LIN {X 0,Y 455.491,Z 844.733,A -85,B 0,C 180,E1 19302.236,E2 19302.236} C_VEL
LIN {X 0,Y 459.84,Z 821.771,A -85,B 0,C 180,E1 19301.253,E2 19301.253} C_VEL
LIN {X 0,Y 463.636,Z 798.381,A -85,B 0,C 180,E1 19300.452,E2 19300.452} C_VEL
LIN {X 0,Y 466.606,Z 774.028,A -85,B 0,C 180,E1 19299.835,E2 19299.835} C_VEL
LIN {X 0,Y 468.518,Z 750.577,A -85,B 0,C 180,E1 19299.385,E2 19299.385} C_VEL
LIN {X 0,Y 481.73,Z 500.688,A -85,B 0,C 180,E1 19295.435,E2 19295.435} C_VEL
LIN {X 0,Y 482.067,Z 491.701,A -85,B 0,C 180,E1 19295.268,E2 19295.268} C_VEL
LIN {X 0,Y 472.219,Z 474.079,A -85,B 0,C 180,E1 19293.15,E2 19293.15} C_VEL
LIN {X 0,Y 462.43,Z 457.753,A -85,B 0,C 180,E1 19290.861,E2 19290.861} C_VEL
LIN {X 0,Y 452.462,Z 442.354,A -85,B 0,C 180,E1 19288.296,E2 19288.296} C_VEL
LIN {X 0,Y 445.961,Z 432.998,A -85,B 0,C 180,E1 19286.463,E2 19286.463} C_VEL
LIN {X 0,Y 439.102,Z 423.302,A -85,B 0,C 180,E1 19284.341,E2 19284.341} C_VEL
LIN {X 0,Y 433.648,Z 416.334,A -85,B 0,C 180,E1 19282.505,E2 19282.505} C_VEL
LIN {X 0,Y 429.886,Z 411.664,A -85,B 0,C 180,E1 19281.132,E2 19281.132} C_VEL
LIN {X 0,Y 425.512,Z 406.796,A -85,B 0,C 180,E1 19279.421,E2 19279.421} C_VEL
LIN {X 0,Y 424.17,Z 404.903,A -85,B 0,C 180,E1 19278.841,E2 19278.841} C_VEL
LIN {X 0,Y 420.773,Z 401.5,A -85,B 0,C 180,E1 19277.351,E2 19277.351} C_VEL
LIN {X 0,Y 419.067,Z 398.833,A -85,B 0,C 180,E1 19276.495,E2 19276.495} C_VEL
LIN {X 0,Y 415.64,Z 396.018,A -85,B 0,C 180,E1 19274.774,E2 19274.774} C_VEL
LIN {X 0,Y 413.682,Z 392.463,A -85,B 0,C 180,E1 19273.56,E2 19273.56} C_VEL
LIN {X 0,Y 409.982,Z 390.014,A -85,B 0,C 180,E1 19271.251,E2 19271.251} C_VEL
LIN {X 0,Y 408.148,Z 386.758,A -85,B 0,C 180,E1 19269.732,E2 19269.732} C_VEL
LIN {X 0,Y 407.71,Z 385.774,A -85,B 0,C 180,E1 19269.315,E2 19269.315} C_VEL
LIN {X 0,Y 403.812,Z 383.595,A -85,B 0,C 180,E1 19265.399,E2 19265.399} C_VEL
LIN {X 0,Y 401.716,Z 379.418,A -85,B 0,C 180,E1 19259.857,E2 19259.857} C_VEL
LIN {X 0,Y 401.699,Z 379.301,A -85,B 0,C 180,E1 19258.003,E2 19258.003} C_VEL
LIN {X 0,Y 402.926,Z 382.497,A -85,B 0,C 180,E1 19253.588,E2 19253.588} C_VEL
LIN {X 0,Y 406.71,Z 385.47,A -85,B 0,C 180,E1 19249.088,E2 19249.088} C_VEL
LIN {X 0,Y 407.878,Z 386.044,A -85,B 0,C 180,E1 19248.116,E2 19248.116} C_VEL
LIN {X 0,Y 409.365,Z 389.184,A -85,B 0,C 180,E1 19246.798,E2 19246.798} C_VEL
LIN {X 0,Y 412.3,Z 391.844,A -85,B 0,C 180,E1 19244.816,E2 19244.816} C_VEL
LIN {X 0,Y 413.753,Z 392.667,A -85,B 0,C 180,E1 19243.972,E2 19243.972} C_VEL
LIN {X 0,Y 416.055,Z 396.475,A -85,B 0,C 180,E1 19242.583,E2 19242.583} C_VEL
LIN {X 0,Y 419.443,Z 399.307,A -85,B 0,C 180,E1 19240.902,E2 19240.902} C_VEL
LIN {X 0,Y 422.238,Z 403.299,A -85,B 0,C 180,E1 19239.556,E2 19239.556} C_VEL
LIN {X 0,Y 424.839,Z 405.657,A -85,B 0,C 180,E1 19238.459,E2 19238.459} C_VEL
LIN {X 0,Y 428.113,Z 409.894,A -85,B 0,C 180,E1 19237.115,E2 19237.115} C_VEL
LIN {X 0,Y 430.045,Z 411.854,A -85,B 0,C 180,E1 19236.391,E2 19236.391} C_VEL
LIN {X 0,Y 433.924,Z 416.564,A -85,B 0,C 180,E1 19234.986,E2 19234.986} C_VEL
LIN {X 0,Y 439.996,Z 424.177,A -85,B 0,C 180,E1 19232.967,E2 19232.967} C_VEL
LIN {X 0,Y 444.51,Z 429.966,A -85,B 0,C 180,E1 19231.585,E2 19231.585} C_VEL
LIN {X 0,Y 451.641,Z 439.191,A -85,B 0,C 180,E1 19229.573,E2 19229.573} C_VEL
LIN {X 0,Y 461.95,Z 453.355,A -85,B 0,C 180,E1 19226.944,E2 19226.944} C_VEL
LIN {X 0,Y 473.346,Z 470.153,A -85,B 0,C 180,E1 19224.337,E2 19224.337} C_VEL
LIN {X 0,Y 482.433,Z 484.639,A -85,B 0,C 180,E1 19222.43,E2 19222.43} C_VEL
LIN {X 0,Y 468.967,Z 736.517,A -85,B 0,C 180,E1 19218.449,E2 19218.449} C_VEL
LIN {X 0,Y 467.166,Z 758.61,A -85,B 0,C 180,E1 19218.013,E2 19218.013} C_VEL
LIN {X 0,Y 464.253,Z 783.344,A -85,B 0,C 180,E1 19217.35,E2 19217.35} C_VEL
LIN {X 0,Y 460.975,Z 804.43,A -85,B 0,C 180,E1 19216.605,E2 19216.605} C_VEL
LIN {X 0,Y 457.064,Z 825.889,A -85,B 0,C 180,E1 19215.672,E2 19215.672} C_VEL
LIN {X 0,Y 452.059,Z 849.09,A -85,B 0,C 180,E1 19214.422,E2 19214.422} C_VEL
LIN {X 0,Y 447.255,Z 868.657,A -85,B 0,C 180,E1 19213.165,E2 19213.165} C_VEL
LIN {X 0,Y 441.166,Z 891.084,A -85,B 0,C 180,E1 19211.438,E2 19211.438} C_VEL
LIN {X 0,Y 435.995,Z 908.438,A -85,B 0,C 180,E1 19209.866,E2 19209.866} C_VEL
LIN {X 0,Y 429.83,Z 928.005,A -85,B 0,C 180,E1 19207.804,E2 19207.804} C_VEL
LIN {X 0,Y 424.092,Z 945.022,A -85,B 0,C 180,E1 19205.687,E2 19205.687} C_VEL
LIN {X 0,Y 418.144,Z 962.284,A -85,B 0,C 180,E1 19203.202,E2 19203.202} C_VEL
LIN {X 0,Y 412.713,Z 977.598,A -85,B 0,C 180,E1 19200.582,E2 19200.582} C_VEL
LIN {X 0,Y 407.773,Z 991.832,A -85,B 0,C 180,E1 19197.768,E2 19197.768} C_VEL
LIN {X 0,Y 403.388,Z 1004.565,A -85,B 0,C 180,E1 19194.765,E2 19194.765} C_VEL
LIN {X 0,Y 399.844,Z 1015.636,A -85,B 0,C 180,E1 19191.722,E2 19191.722} C_VEL
LIN {X 0,Y 396.862,Z 1025.775,A -85,B 0,C 180,E1 19188.357,E2 19188.357} C_VEL
LIN {X 0,Y 394.876,Z 1033.558,A -85,B 0,C 180,E1 19185.256,E2 19185.256} C_VEL
LIN {X 0,Y 393.323,Z 1040.946,A -85,B 0,C 180,E1 19181.586,E2 19181.586} C_VEL
LIN {X 0,Y 392.551,Z 1045.732,A -85,B 0,C 180,E1 19178.496,E2 19178.496} C_VEL
LIN {X 0,Y 392.145,Z 1049.646,A -85,B 0,C 180,E1 19175.12,E2 19175.12} C_VEL
LIN {X 0,Y 391.997,Z 1051.962,A -85,B 0,C 180,E1 19171.754,E2 19171.754} C_VEL
LIN {X 0,Y 391.965,Z 1052.864,A -85,B 0,C 180,E1 19168.977,E2 19168.977} C_VEL
LIN {X 0,Y 391.973,Z 1052.777,A -85,B 0,C 180,E1 19165.904,E2 19165.904} C_VEL
LIN {X 0,Y 392.058,Z 1051.214,A -85,B 0,C 180,E1 19162.379,E2 19162.379} C_VEL
LIN {X 0,Y 392.307,Z 1048.524,A -85,B 0,C 180,E1 19159.277,E2 19159.277} C_VEL
LIN {X 0,Y 392.861,Z 1044.661,A -85,B 0,C 180,E1 19156.158,E2 19156.158} C_VEL
LIN {X 0,Y 393.592,Z 1040.768,A -85,B 0,C 180,E1 19153.731,E2 19153.731} C_VEL
LIN {X 0,Y 393.032,Z 1038.922,A -85,B 0,C 180,E1 19152.636,E2 19152.636} C_VEL
LIN {X 0,Y 388.297,Z 1033.538,A -85,B 0,C 180,E1 19149.698,E2 19149.698} C_VEL
LIN {X 0,Y 388.161,Z 1031.488,A -85,B 0,C 180,E1 19148.76,E2 19148.76} C_VEL
LIN {X 0,Y 391.208,Z 1021.724,A -85,B 0,C 180,E1 19145.057,E2 19145.057} C_VEL
LIN {X 0,Y 394.53,Z 1012.11,A -85,B 0,C 180,E1 19142.04,E2 19142.04} C_VEL
LIN {X 0,Y 399.372,Z 999.124,A -85,B 0,C 180,E1 19138.617,E2 19138.617} C_VEL
LIN {X 0,Y 404.183,Z 986.584,A -85,B 0,C 180,E1 19135.836,E2 19135.836} C_VEL
LIN {X 0,Y 410.106,Z 971.471,A -85,B 0,C 180,E1 19132.971,E2 19132.971} C_VEL
LIN {X 0,Y 416.021,Z 956.003,A -85,B 0,C 180,E1 19130.49,E2 19130.49} C_VEL
LIN {X 0,Y 422.663,Z 938.384,A -85,B 0,C 180,E1 19128.063,E2 19128.063} C_VEL
LIN {X 0,Y 428.961,Z 920.629,A -85,B 0,C 180,E1 19126.003,E2 19126.003} C_VEL
LIN {X 0,Y 435.548,Z 901.209,A -85,B 0,C 180,E1 19124.065,E2 19124.065} C_VEL
LIN {X 0,Y 441.835,Z 880.625,A -85,B 0,C 180,E1 19122.35,E2 19122.35} C_VEL
LIN {X 0,Y 447.423,Z 860.804,A -85,B 0,C 180,E1 19120.944,E2 19120.944} C_VEL
LIN {X 0,Y 453.017,Z 838.232,A -85,B 0,C 180,E1 19119.619,E2 19119.619} C_VEL
LIN {X 0,Y 457.191,Z 818.895,A -85,B 0,C 180,E1 19118.669,E2 19118.669} C_VEL
LIN {X 0,Y 461.767,Z 793.938,A -85,B 0,C 180,E1 19117.68,E2 19117.68} C_VEL
LIN {X 0,Y 464.905,Z 772.264,A -85,B 0,C 180,E1 19117.014,E2 19117.014} C_VEL
LIN {X 0,Y 467.655,Z 747.34,A -85,B 0,C 180,E1 19116.439,E2 19116.439} C_VEL
LIN {X 0,Y 471.279,Z 687.121,A -85,B 0,C 180,E1 19115.457,E2 19115.457} C_VEL
LIN {X 0,Y 482.561,Z 491.611,A -85,B 0,C 180,E1 19112.355,E2 19112.355} C_VEL
LIN {X 0,Y 471.614,Z 474.658,A -85,B 0,C 180,E1 19109.778,E2 19109.778} C_VEL
LIN {X 0,Y 462.04,Z 460.876,A -85,B 0,C 180,E1 19107.274,E2 19107.274} C_VEL
LIN {X 0,Y 454.319,Z 450.447,A -85,B 0,C 180,E1 19105.032,E2 19105.032} C_VEL
LIN {X 0,Y 447.642,Z 441.602,A -85,B 0,C 180,E1 19102.871,E2 19102.871} C_VEL
LIN {X 0,Y 443.202,Z 436.029,A -85,B 0,C 180,E1 19101.299,E2 19101.299} C_VEL
LIN {X 0,Y 439.218,Z 430.987,A -85,B 0,C 180,E1 19099.759,E2 19099.759} C_VEL
LIN {X 0,Y 435.448,Z 426.19,A -85,B 0,C 180,E1 19098.163,E2 19098.163} C_VEL
LIN {X 0,Y 431.395,Z 421.665,A -85,B 0,C 180,E1 19096.287,E2 19096.287} C_VEL
LIN {X 0,Y 430.163,Z 419.832,A -85,B 0,C 180,E1 19095.643,E2 19095.643} C_VEL
LIN {X 0,Y 426.685,Z 416.352,A -85,B 0,C 180,E1 19093.76,E2 19093.76} C_VEL
LIN {X 0,Y 425.161,Z 413.779,A -85,B 0,C 180,E1 19092.772,E2 19092.772} C_VEL
LIN {X 0,Y 421.812,Z 411.007,A -85,B 0,C 180,E1 19090.517,E2 19090.517} C_VEL
LIN {X 0,Y 419.877,Z 407.432,A -85,B 0,C 180,E1 19088.767,E2 19088.767} C_VEL
LIN {X 0,Y 415.834,Z 404.429,A -85,B 0,C 180,E1 19083.999,E2 19083.999} C_VEL
LIN {X 0,Y 414.742,Z 401.753,A -85,B 0,C 180,E1 19080.138,E2 19080.138} C_VEL
LIN {X 0,Y 414.717,Z 401.619,A -85,B 0,C 180,E1 19078.618,E2 19078.618} C_VEL
LIN {X 0,Y 415.242,Z 403.337,A -85,B 0,C 180,E1 19075.719,E2 19075.719} C_VEL
LIN {X 0,Y 419.25,Z 407.195,A -85,B 0,C 180,E1 19070.112,E2 19070.112} C_VEL
LIN {X 0,Y 420.088,Z 407.737,A -85,B 0,C 180,E1 19069.37,E2 19069.37} C_VEL
LIN {X 0,Y 422.241,Z 411.567,A -85,B 0,C 180,E1 19067.486,E2 19067.486} C_VEL
LIN {X 0,Y 425.517,Z 414.256,A -85,B 0,C 180,E1 19065.333,E2 19065.333} C_VEL
LIN {X 0,Y 428.154,Z 418.196,A -85,B 0,C 180,E1 19063.725,E2 19063.725} C_VEL
LIN {X 0,Y 430.667,Z 420.442,A -85,B 0,C 180,E1 19062.433,E2 19062.433} C_VEL
LIN {X 0,Y 434.083,Z 424.878,A -85,B 0,C 180,E1 19060.768,E2 19060.768} C_VEL
LIN {X 0,Y 435.806,Z 426.713,A -85,B 0,C 180,E1 19060.01,E2 19060.01} C_VEL
LIN {X 0,Y 439.552,Z 431.305,A -85,B 0,C 180,E1 19058.446,E2 19058.446} C_VEL
LIN {X 0,Y 446.538,Z 441.039,A -85,B 0,C 180,E1 19055.809,E2 19055.809} C_VEL
LIN {X 0,Y 454.673,Z 452.672,A -85,B 0,C 180,E1 19053.133,E2 19053.133} C_VEL
LIN {X 0,Y 464.779,Z 468.395,A -85,B 0,C 180,E1 19050.201,E2 19050.201} C_VEL
LIN {X 0,Y 473.883,Z 483.545,A -85,B 0,C 180,E1 19047.842,E2 19047.842} C_VEL
LIN {X 0,Y 482.418,Z 498.724,A -85,B 0,C 180,E1 19045.816,E2 19045.816} C_VEL
LIN {X 0,Y 468.053,Z 748.938,A -85,B 0,C 180,E1 19041.855,E2 19041.855} C_VEL
LIN {X 0,Y 465.972,Z 773.134,A -85,B 0,C 180,E1 19041.396,E2 19041.396} C_VEL
LIN {X 0,Y 462.858,Z 797.389,A -85,B 0,C 180,E1 19040.795,E2 19040.795} C_VEL
LIN {X 0,Y 458.752,Z 821.123,A -85,B 0,C 180,E1 19039.997,E2 19039.997} C_VEL
LIN {X 0,Y 454.683,Z 841.259,A -85,B 0,C 180,E1 19039.156,E2 19039.156} C_VEL
LIN {X 0,Y 449.116,Z 864.849,A -85,B 0,C 180,E1 19037.934,E2 19037.934} C_VEL
LIN {X 0,Y 444.065,Z 883.795,A -85,B 0,C 180,E1 19036.754,E2 19036.754} C_VEL
LIN {X 0,Y 437.897,Z 904.941,A -85,B 0,C 180,E1 19035.198,E2 19035.198} C_VEL
LIN {X 0,Y 431.615,Z 924.469,A -85,B 0,C 180,E1 19033.475,E2 19033.475} C_VEL
LIN {X 0,Y 425.219,Z 943.337,A -85,B 0,C 180,E1 19031.538,E2 19031.538} C_VEL
LIN {X 0,Y 418.497,Z 961.862,A -85,B 0,C 180,E1 19029.275,E2 19029.275} C_VEL
LIN {X 0,Y 412.462,Z 978.197,A -85,B 0,C 180,E1 19026.956,E2 19026.956} C_VEL
LIN {X 0,Y 406.308,Z 994.527,A -85,B 0,C 180,E1 19024.221,E2 19024.221} C_VEL
LIN {X 0,Y 401.467,Z 1007.481,A -85,B 0,C 180,E1 19021.703,E2 19021.703} C_VEL
LIN {X 0,Y 396.129,Z 1022.244,A -85,B 0,C 180,E1 19018.329,E2 19018.329} C_VEL
LIN {X 0,Y 392.382,Z 1033.25,A -85,B 0,C 180,E1 19015.348,E2 19015.348} C_VEL
LIN {X 0,Y 388.944,Z 1044.487,A -85,B 0,C 180,E1 19011.727,E2 19011.727} C_VEL
LIN {X 0,Y 386.8,Z 1052.635,A -85,B 0,C 180,E1 19008.54,E2 19008.54} C_VEL
LIN {X 0,Y 385.198,Z 1060.295,A -85,B 0,C 180,E1 19004.891,E2 19004.891} C_VEL
LIN {X 0,Y 384.382,Z 1065.649,A -85,B 0,C 180,E1 19001.554,E2 19001.554} C_VEL
LIN {X 0,Y 384.037,Z 1069.516,A -85,B 0,C 180,E1 18998.384,E2 18998.384} C_VEL
LIN {X 0,Y 383.949,Z 1072.401,A -85,B 0,C 180,E1 18994.78,E2 18994.78} C_VEL
LIN {X 0,Y 383.953,Z 1073.541,A -85,B 0,C 180,E1 18991.642,E2 18991.642} C_VEL
LIN {X 0,Y 383.963,Z 1073.547,A -85,B 0,C 180,E1 18988.806,E2 18988.806} C_VEL
LIN {X 0,Y 383.948,Z 1072.419,A -85,B 0,C 180,E1 18985.669,E2 18985.669} C_VEL
LIN {X 0,Y 384.004,Z 1069.534,A -85,B 0,C 180,E1 18982.068,E2 18982.068} C_VEL
LIN {X 0,Y 384.28,Z 1065.866,A -85,B 0,C 180,E1 18979.05,E2 18979.05} C_VEL
LIN {X 0,Y 384.979,Z 1060.531,A -85,B 0,C 180,E1 18975.715,E2 18975.715} C_VEL
LIN {X 0,Y 386.406,Z 1052.891,A -85,B 0,C 180,E1 18972.065,E2 18972.065} C_VEL
LIN {X 0,Y 388.362,Z 1044.717,A -85,B 0,C 180,E1 18968.872,E2 18968.872} C_VEL
LIN {X 0,Y 391.549,Z 1033.43,A -85,B 0,C 180,E1 18965.241,E2 18965.241} C_VEL
LIN {X 0,Y 394.875,Z 1022.921,A -85,B 0,C 180,E1 18962.394,E2 18962.394} C_VEL
LIN {X 0,Y 399.705,Z 1008.63,A -85,B 0,C 180,E1 18959.098,E2 18959.098} C_VEL
LIN {X 0,Y 404.296,Z 995.515,A -85,B 0,C 180,E1 18956.529,E2 18956.529} C_VEL
LIN {X 0,Y 409.981,Z 979.623,A -85,B 0,C 180,E1 18953.828,E2 18953.828} C_VEL
LIN {X 0,Y 415.936,Z 962.527,A -85,B 0,C 180,E1 18951.379,E2 18951.379} C_VEL
LIN {X 0,Y 422.291,Z 944.111,A -85,B 0,C 180,E1 18949.104,E2 18949.104} C_VEL
LIN {X 0,Y 428.466,Z 924.968,A -85,B 0,C 180,E1 18947.119,E2 18947.119} C_VEL
LIN {X 0,Y 434.363,Z 905.758,A -85,B 0,C 180,E1 18945.404,E2 18945.404} C_VEL
LIN {X 0,Y 440.427,Z 884.078,A -85,B 0,C 180,E1 18943.785,E2 18943.785} C_VEL
LIN {X 0,Y 445.338,Z 864.832,A -85,B 0,C 180,E1 18942.571,E2 18942.571} C_VEL
LIN {X 0,Y 450.75,Z 840.786,A -85,B 0,C 180,E1 18941.316,E2 18941.316} C_VEL
LIN {X 0,Y 454.679,Z 820.431,A -85,B 0,C 180,E1 18940.457,E2 18940.457} C_VEL
LIN {X 0,Y 458.627,Z 796.402,A -85,B 0,C 180,E1 18939.647,E2 18939.647} C_VEL
LIN {X 0,Y 461.517,Z 772.739,A -85,B 0,C 180,E1 18939.057,E2 18939.057} C_VEL
LIN {X 0,Y 463.533,Z 747.792,A -85,B 0,C 180,E1 18938.583,E2 18938.583} C_VEL
LIN {X 0,Y 477.177,Z 497.517,A -85,B 0,C 180,E1 18934.61,E2 18934.61} C_VEL
LIN {X 0,Y 477.146,Z 495.381,A -85,B 0,C 180,E1 18934.551,E2 18934.551} C_VEL
LIN {X 0,Y 468.133,Z 479.157,A -85,B 0,C 180,E1 18932.547,E2 18932.547} C_VEL
LIN {X 0,Y 458.488,Z 462.849,A -85,B 0,C 180,E1 18930.214,E2 18930.214} C_VEL
LIN {X 0,Y 448.517,Z 447.367,A -85,B 0,C 180,E1 18927.554,E2 18927.554} C_VEL
LIN {X 0,Y 440.843,Z 436.152,A -85,B 0,C 180,E1 18925.276,E2 18925.276} C_VEL
LIN {X 0,Y 435.436,Z 428.576,A -85,B 0,C 180,E1 18923.515,E2 18923.515} C_VEL
LIN {X 0,Y 431.436,Z 423.529,A -85,B 0,C 180,E1 18922.124,E2 18922.124} C_VEL
LIN {X 0,Y 427.082,Z 418.165,A -85,B 0,C 180,E1 18920.488,E2 18920.488} C_VEL
LIN {X 0,Y 423.465,Z 413.928,A -85,B 0,C 180,E1 18919.017,E2 18919.017} C_VEL
LIN {X 0,Y 422.283,Z 412.371,A -85,B 0,C 180,E1 18918.499,E2 18918.499} C_VEL
LIN {X 0,Y 418.833,Z 408.657,A -85,B 0,C 180,E1 18916.933,E2 18916.933} C_VEL
LIN {X 0,Y 417.554,Z 406.557,A -85,B 0,C 180,E1 18916.271,E2 18916.271} C_VEL
LIN {X 0,Y 414.063,Z 403.556,A -85,B 0,C 180,E1 18914.474,E2 18914.474} C_VEL
LIN {X 0,Y 412.008,Z 400.163,A -85,B 0,C 180,E1 18913.187,E2 18913.187} C_VEL
LIN {X 0,Y 408.446,Z 397.48,A -85,B 0,C 180,E1 18910.865,E2 18910.865} C_VEL
LIN {X 0,Y 406.632,Z 393.911,A -85,B 0,C 180,E1 18909.269,E2 18909.269} C_VEL
LIN {X 0,Y 402.105,Z 390.661,A -85,B 0,C 180,E1 18904.278,E2 18904.278} C_VEL
LIN {X 0,Y 400.727,Z 387.333,A -85,B 0,C 180,E1 18899.714,E2 18899.714} C_VEL
LIN {X 0,Y 400.721,Z 387.274,A -85,B 0,C 180,E1 18897.998,E2 18897.998} C_VEL
LIN {X 0,Y 401.95,Z 390.495,A -85,B 0,C 180,E1 18893.573,E2 18893.573} C_VEL
LIN {X 0,Y 405.751,Z 393.425,A -85,B 0,C 180,E1 18889.062,E2 18889.062} C_VEL
LIN {X 0,Y 406.606,Z 393.952,A -85,B 0,C 180,E1 18888.331,E2 18888.331} C_VEL
LIN {X 0,Y 408.39,Z 397.344,A -85,B 0,C 180,E1 18886.766,E2 18886.766} C_VEL
LIN {X 0,Y 411.352,Z 399.841,A -85,B 0,C 180,E1 18884.78,E2 18884.78} C_VEL
LIN {X 0,Y 412.319,Z 400.519,A -85,B 0,C 180,E1 18884.204,E2 18884.204} C_VEL
LIN {X 0,Y 414.954,Z 404.57,A -85,B 0,C 180,E1 18882.615,E2 18882.615} C_VEL
LIN {X 0,Y 417.856,Z 407.066,A -85,B 0,C 180,E1 18881.153,E2 18881.153} C_VEL
LIN {X 0,Y 420.843,Z 411.141,A -85,B 0,C 180,E1 18879.703,E2 18879.703} C_VEL
LIN {X 0,Y 423.031,Z 413.181,A -85,B 0,C 180,E1 18878.763,E2 18878.763} C_VEL
LIN {X 0,Y 426.507,Z 417.6,A -85,B 0,C 180,E1 18877.316,E2 18877.316} C_VEL
LIN {X 0,Y 428.237,Z 419.511,A -85,B 0,C 180,E1 18876.65,E2 18876.65} C_VEL
LIN {X 0,Y 433.3,Z 425.813,A -85,B 0,C 180,E1 18874.801,E2 18874.801} C_VEL
LIN {X 0,Y 438.073,Z 431.845,A -85,B 0,C 180,E1 18873.206,E2 18873.206} C_VEL
LIN {X 0,Y 444.947,Z 440.653,A -85,B 0,C 180,E1 18871.108,E2 18871.108} C_VEL
LIN {X 0,Y 455.338,Z 454.837,A -85,B 0,C 180,E1 18868.269,E2 18868.269} C_VEL
LIN {X 0,Y 465.733,Z 470.04,A -85,B 0,C 180,E1 18865.734,E2 18865.734} C_VEL
LIN {X 0,Y 476.542,Z 486.919,A -85,B 0,C 180,E1 18863.348,E2 18863.348} C_VEL
LIN {X 0,Y 477.491,Z 488.857,A -85,B 0,C 180,E1 18863.139,E2 18863.139} C_VEL
LIN {X 0,Y 463.742,Z 737.798,A -85,B 0,C 180,E1 18859.183,E2 18859.183} C_VEL
LIN {X 0,Y 461.889,Z 759.635,A -85,B 0,C 180,E1 18858.746,E2 18858.746} C_VEL
LIN {X 0,Y 458.714,Z 785.283,A -85,B 0,C 180,E1 18858.042,E2 18858.042} C_VEL
LIN {X 0,Y 455.408,Z 805.842,A -85,B 0,C 180,E1 18857.305,E2 18857.305} C_VEL
LIN {X 0,Y 451.039,Z 828.996,A -85,B 0,C 180,E1 18856.277,E2 18856.277} C_VEL
LIN {X 0,Y 446.157,Z 850.517,A -85,B 0,C 180,E1 18855.088,E2 18855.088} C_VEL
LIN {X 0,Y 440.981,Z 870.936,A -85,B 0,C 180,E1 18853.754,E2 18853.754} C_VEL
LIN {X 0,Y 434.94,Z 892.259,A -85,B 0,C 180,E1 18852.077,E2 18852.077} C_VEL
LIN {X 0,Y 429.623,Z 909.526,A -85,B 0,C 180,E1 18850.491,E2 18850.491} C_VEL
LIN {X 0,Y 422.879,Z 930.049,A -85,B 0,C 180,E1 18848.278,E2 18848.278} C_VEL
LIN {X 0,Y 417.38,Z 945.825,A -85,B 0,C 180,E1 18846.279,E2 18846.279} C_VEL
LIN {X 0,Y 411.365,Z 962.639,A -85,B 0,C 180,E1 18843.822,E2 18843.822} C_VEL
LIN {X 0,Y 405.72,Z 977.942,A -85,B 0,C 180,E1 18841.167,E2 18841.167} C_VEL
LIN {X 0,Y 400.577,Z 992.163,A -85,B 0,C 180,E1 18838.311,E2 18838.311} C_VEL
LIN {X 0,Y 395.997,Z 1004.877,A -85,B 0,C 180,E1 18835.26,E2 18835.26} C_VEL
LIN {X 0,Y 392.289,Z 1015.938,A -85,B 0,C 180,E1 18832.162,E2 18832.162} C_VEL
LIN {X 0,Y 389.154,Z 1026.06,A -85,B 0,C 180,E1 18828.734,E2 18828.734} C_VEL
LIN {X 0,Y 387.063,Z 1033.804,A -85,B 0,C 180,E1 18825.585,E2 18825.585} C_VEL
LIN {X 0,Y 385.412,Z 1041.204,A -85,B 0,C 180,E1 18821.827,E2 18821.827} C_VEL
LIN {X 0,Y 384.591,Z 1045.982,A -85,B 0,C 180,E1 18818.673,E2 18818.673} C_VEL
LIN {X 0,Y 384.16,Z 1049.886,A -85,B 0,C 180,E1 18815.227,E2 18815.227} C_VEL
LIN {X 0,Y 384.002,Z 1052.187,A -85,B 0,C 180,E1 18811.791,E2 18811.791} C_VEL
LIN {X 0,Y 383.968,Z 1053.081,A -85,B 0,C 180,E1 18808.955,E2 18808.955} C_VEL
LIN {X 0,Y 383.976,Z 1052.987,A -85,B 0,C 180,E1 18805.819,E2 18805.819} C_VEL
LIN {X 0,Y 384.07,Z 1051.41,A -85,B 0,C 180,E1 18802.22,E2 18802.22} C_VEL
LIN {X 0,Y 384.344,Z 1048.714,A -85,B 0,C 180,E1 18799.052,E2 18799.052} C_VEL
LIN {X 0,Y 384.981,Z 1044.641,A -85,B 0,C 180,E1 18795.715,E2 18795.715} C_VEL
LIN {X 0,Y 386.285,Z 1038.504,A -85,B 0,C 180,E1 18792.059,E2 18792.059} C_VEL
LIN {X 0,Y 388.096,Z 1031.703,A -85,B 0,C 180,E1 18788.853,E2 18788.853} C_VEL
LIN {X 0,Y 388.161,Z 1031.488,A -85,B 0,C 180,E1 18788.76,E2 18788.76} C_VEL
LIN {X 0,Y 387.959,Z 1029.057,A -85,B 0,C 180,E1 18787.672,E2 18787.672} C_VEL
LIN {X 0,Y 384.255,Z 1022.305,A -85,B 0,C 180,E1 18784.732,E2 18784.732} C_VEL
LIN {X 0,Y 384.449,Z 1019.742,A -85,B 0,C 180,E1 18783.812,E2 18783.812} C_VEL
LIN {X 0,Y 388.656,Z 1008.562,A -85,B 0,C 180,E1 18780.399,E2 18780.399} C_VEL
LIN {X 0,Y 393.297,Z 996.716,A -85,B 0,C 180,E1 18777.386,E2 18777.386} C_VEL
LIN {X 0,Y 398.824,Z 983.196,A -85,B 0,C 180,E1 18774.434,E2 18774.434} C_VEL
LIN {X 0,Y 404.831,Z 968.184,A -85,B 0,C 180,E1 18771.688,E2 18771.688} C_VEL
LIN {X 0,Y 411.291,Z 952.107,A -85,B 0,C 180,E1 18769.159,E2 18769.159} C_VEL
LIN {X 0,Y 417.998,Z 934.542,A -85,B 0,C 180,E1 18766.832,E2 18766.832} C_VEL
LIN {X 0,Y 423.977,Z 918.218,A -85,B 0,C 180,E1 18764.968,E2 18764.968} C_VEL
LIN {X 0,Y 431.284,Z 896.797,A -85,B 0,C 180,E1 18762.894,E2 18762.894} C_VEL
LIN {X 0,Y 437.077,Z 878.257,A -85,B 0,C 180,E1 18761.379,E2 18761.379} C_VEL
LIN {X 0,Y 443.573,Z 855.296,A -85,B 0,C 180,E1 18759.806,E2 18759.806} C_VEL
LIN {X 0,Y 448.409,Z 835.821,A -85,B 0,C 180,E1 18758.698,E2 18758.698} C_VEL
LIN {X 0,Y 453.294,Z 813.528,A -85,B 0,C 180,E1 18757.637,E2 18757.637} C_VEL
LIN {X 0,Y 457.351,Z 790.629,A -85,B 0,C 180,E1 18756.78,E2 18756.78} C_VEL
LIN {X 0,Y 460.472,Z 769.119,A -85,B 0,C 180,E1 18756.14,E2 18756.14} C_VEL
LIN {X 0,Y 463.129,Z 743.445,A -85,B 0,C 180,E1 18755.581,E2 18755.581} C_VEL
LIN {X 0,Y 477.157,Z 509.888,A -85,B 0,C 180,E1 18751.854,E2 18751.854} C_VEL
LIN {X 0,Y 477.927,Z 495.802,A -85,B 0,C 180,E1 18751.614,E2 18751.614} C_VEL
LIN {X 0,Y 467.87,Z 480.108,A -85,B 0,C 180,E1 18749.161,E2 18749.161} C_VEL
LIN {X 0,Y 458.806,Z 466.914,A -85,B 0,C 180,E1 18746.711,E2 18746.711} C_VEL
LIN {X 0,Y 449.89,Z 454.557,A -85,B 0,C 180,E1 18743.999,E2 18743.999} C_VEL
LIN {X 0,Y 441.733,Z 443.923,A -85,B 0,C 180,E1 18741.164,E2 18741.164} C_VEL
LIN {X 0,Y 437.158,Z 438.224,A -85,B 0,C 180,E1 18739.369,E2 18739.369} C_VEL
LIN {X 0,Y 432.967,Z 432.988,A -85,B 0,C 180,E1 18737.54,E2 18737.54} C_VEL
LIN {X 0,Y 429.53,Z 428.825,A -85,B 0,C 180,E1 18735.874,E2 18735.874} C_VEL
LIN {X 0,Y 428.429,Z 427.355,A -85,B 0,C 180,E1 18735.291,E2 18735.291} C_VEL
LIN {X 0,Y 424.952,Z 423.571,A -85,B 0,C 180,E1 18733.332,E2 18733.332} C_VEL
LIN {X 0,Y 423.763,Z 421.546,A -85,B 0,C 180,E1 18732.538,E2 18732.538} C_VEL
LIN {X 0,Y 420.329,Z 418.472,A -85,B 0,C 180,E1 18730.139,E2 18730.139} C_VEL
LIN {X 0,Y 418.595,Z 415.277,A -85,B 0,C 180,E1 18728.517,E2 18728.517} C_VEL
LIN {X 0,Y 414.654,Z 412.078,A -85,B 0,C 180,E1 18723.595,E2 18723.595} C_VEL
LIN {X 0,Y 413.753,Z 409.569,A -85,B 0,C 180,E1 18719.862,E2 18719.862} C_VEL
LIN {X 0,Y 413.822,Z 409.954,A -85,B 0,C 180,E1 18717.646,E2 18717.646} C_VEL
LIN {X 0,Y 418.138,Z 415.092,A -85,B 0,C 180,E1 18710.225,E2 18710.225} C_VEL
LIN {X 0,Y 418.882,Z 415.623,A -85,B 0,C 180,E1 18709.548,E2 18709.548} C_VEL
LIN {X 0,Y 421.003,Z 419.369,A -85,B 0,C 180,E1 18707.658,E2 18707.658} C_VEL
LIN {X 0,Y 424.072,Z 421.923,A -85,B 0,C 180,E1 18705.596,E2 18705.596} C_VEL
LIN {X 0,Y 426.834,Z 426.008,A -85,B 0,C 180,E1 18703.883,E2 18703.883} C_VEL
LIN {X 0,Y 429.181,Z 428.229,A -85,B 0,C 180,E1 18702.65,E2 18702.65} C_VEL
LIN {X 0,Y 432.702,Z 432.705,A -85,B 0,C 180,E1 18700.914,E2 18700.914} C_VEL
LIN {X 0,Y 434.181,Z 434.42,A -85,B 0,C 180,E1 18700.248,E2 18700.248} C_VEL
LIN {X 0,Y 438.948,Z 440.495,A -85,B 0,C 180,E1 18698.239,E2 18698.239} C_VEL
LIN {X 0,Y 444.689,Z 448.712,A -85,B 0,C 180,E1 18696.055,E2 18696.055} C_VEL
LIN {X 0,Y 452.263,Z 459.705,A -85,B 0,C 180,E1 18693.51,E2 18693.51} C_VEL
LIN {X 0,Y 462.215,Z 475.454,A -85,B 0,C 180,E1 18690.554,E2 18690.554} C_VEL
LIN {X 0,Y 471.304,Z 490.869,A -85,B 0,C 180,E1 18688.147,E2 18688.147} C_VEL
LIN {X 0,Y 477.792,Z 502.788,A -85,B 0,C 180,E1 18686.555,E2 18686.555} C_VEL
LIN {X 0,Y 463.026,Z 751.514,A -85,B 0,C 180,E1 18682.597,E2 18682.597} C_VEL
LIN {X 0,Y 460.977,Z 774.068,A -85,B 0,C 180,E1 18682.162,E2 18682.162} C_VEL
LIN {X 0,Y 457.627,Z 798.83,A -85,B 0,C 180,E1 18681.535,E2 18681.535} C_VEL
LIN {X 0,Y 453.795,Z 820.475,A -85,B 0,C 180,E1 18680.804,E2 18680.804} C_VEL
LIN {X 0,Y 449.461,Z 841.373,A -85,B 0,C 180,E1 18679.932,E2 18679.932} C_VEL
LIN {X 0,Y 443.769,Z 864.79,A -85,B 0,C 180,E1 18678.715,E2 18678.715} C_VEL
LIN {X 0,Y 438.553,Z 883.81,A -85,B 0,C 180,E1 18677.525,E2 18677.525} C_VEL
LIN {X 0,Y 431.836,Z 906.004,A -85,B 0,C 180,E1 18675.872,E2 18675.872} C_VEL
LIN {X 0,Y 425.724,Z 924.421,A -85,B 0,C 180,E1 18674.231,E2 18674.231} C_VEL
LIN {X 0,Y 418.908,Z 943.868,A -85,B 0,C 180,E1 18672.215,E2 18672.215} C_VEL
LIN {X 0,Y 412.181,Z 961.726,A -85,B 0,C 180,E1 18670.005,E2 18670.005} C_VEL
LIN {X 0,Y 405.9,Z 978.095,A -85,B 0,C 180,E1 18667.656,E2 18667.656} C_VEL
LIN {X 0,Y 399.636,Z 994.038,A -85,B 0,C 180,E1 18664.957,E2 18664.957} C_VEL
LIN {X 0,Y 394.447,Z 1007.349,A -85,B 0,C 180,E1 18662.335,E2 18662.335} C_VEL
LIN {X 0,Y 388.853,Z 1022.095,A -85,B 0,C 180,E1 18658.909,E2 18658.909} C_VEL
LIN {X 0,Y 384.923,Z 1033.094,A -85,B 0,C 180,E1 18655.875,E2 18655.875} C_VEL
LIN {X 0,Y 381.161,Z 1044.727,A -85,B 0,C 180,E1 18652.032,E2 18652.032} C_VEL
LIN {X 0,Y 378.92,Z 1052.817,A -85,B 0,C 180,E1 18648.78,E2 18648.78} C_VEL
LIN {X 0,Y 377.195,Z 1060.626,A -85,B 0,C 180,E1 18644.9,E2 18644.9} C_VEL
LIN {X 0,Y 376.396,Z 1065.668,A -85,B 0,C 180,E1 18641.648,E2 18641.648} C_VEL
LIN {X 0,Y 376.025,Z 1069.646,A -85,B 0,C 180,E1 18638.256,E2 18638.256} C_VEL
LIN {X 0,Y 375.948,Z 1072.336,A -85,B 0,C 180,E1 18634.576,E2 18634.576} C_VEL
LIN {X 0,Y 375.957,Z 1073.33,A -85,B 0,C 180,E1 18631.676,E2 18631.676} C_VEL
LIN {X 0,Y 375.965,Z 1073.331,A -85,B 0,C 180,E1 18628.781,E2 18628.781} C_VEL
LIN {X 0,Y 375.951,Z 1072.197,A -85,B 0,C 180,E1 18625.576,E2 18625.576} C_VEL
LIN {X 0,Y 376.015,Z 1069.299,A -85,B 0,C 180,E1 18621.898,E2 18621.898} C_VEL
LIN {X 0,Y 376.313,Z 1065.625,A -85,B 0,C 180,E1 18618.816,E2 18618.816} C_VEL
LIN {X 0,Y 377.065,Z 1060.282,A -85,B 0,C 180,E1 18615.409,E2 18615.409} C_VEL
LIN {X 0,Y 378.591,Z 1052.628,A -85,B 0,C 180,E1 18611.682,E2 18611.682} C_VEL
LIN {X 0,Y 380.669,Z 1044.446,A -85,B 0,C 180,E1 18608.424,E2 18608.424} C_VEL
LIN {X 0,Y 384.037,Z 1033.144,A -85,B 0,C 180,E1 18604.723,E2 18604.723} C_VEL
LIN {X 0,Y 387.534,Z 1022.627,A -85,B 0,C 180,E1 18601.825,E2 18601.825} C_VEL
LIN {X 0,Y 392.523,Z 1008.535,A -85,B 0,C 180,E1 18598.52,E2 18598.52} C_VEL
LIN {X 0,Y 397.395,Z 995.196,A -85,B 0,C 180,E1 18595.869,E2 18595.869} C_VEL
LIN {X 0,Y 403.31,Z 979.283,A -85,B 0,C 180,E1 18593.132,E2 18593.132} C_VEL
LIN {X 0,Y 409.632,Z 961.81,A -85,B 0,C 180,E1 18590.606,E2 18590.606} C_VEL
LIN {X 0,Y 416.292,Z 943.126,A -85,B 0,C 180,E1 18588.293,E2 18588.293} C_VEL
LIN {X 0,Y 422.435,Z 924.703,A -85,B 0,C 180,E1 18586.372,E2 18586.372} C_VEL
LIN {X 0,Y 428.561,Z 905.351,A -85,B 0,C 180,E1 18584.634,E2 18584.634} C_VEL
LIN {X 0,Y 434.811,Z 883.629,A -85,B 0,C 180,E1 18583.007,E2 18583.007} C_VEL
LIN {X 0,Y 439.864,Z 864.356,A -85,B 0,C 180,E1 18581.789,E2 18581.789} C_VEL
LIN {X 0,Y 445.381,Z 840.47,A -85,B 0,C 180,E1 18580.541,E2 18580.541} C_VEL
LIN {X 0,Y 449.404,Z 820.168,A -85,B 0,C 180,E1 18579.684,E2 18579.684} C_VEL
LIN {X 0,Y 453.43,Z 796.266,A -85,B 0,C 180,E1 18578.877,E2 18578.877} C_VEL
LIN {X 0,Y 456.393,Z 772.597,A -85,B 0,C 180,E1 18578.286,E2 18578.286} C_VEL
LIN {X 0,Y 458.46,Z 747.708,A -85,B 0,C 180,E1 18577.811,E2 18577.811} C_VEL
LIN {X 0,Y 472.43,Z 499.373,A -85,B 0,C 180,E1 18573.85,E2 18573.85} C_VEL
LIN {X 0,Y 462.964,Z 482.094,A -85,B 0,C 180,E1 18571.656,E2 18571.656} C_VEL
LIN {X 0,Y 452.861,Z 465.203,A -85,B 0,C 180,E1 18569.098,E2 18569.098} C_VEL
LIN {X 0,Y 442.865,Z 449.591,A -85,B 0,C 180,E1 18566.265,E2 18566.265} C_VEL
LIN {X 0,Y 433.988,Z 436.811,A -85,B 0,C 180,E1 18563.418,E2 18563.418} C_VEL
LIN {X 0,Y 429.245,Z 430.714,A -85,B 0,C 180,E1 18561.739,E2 18561.739} C_VEL
LIN {X 0,Y 424.967,Z 425.414,A -85,B 0,C 180,E1 18560.092,E2 18560.092} C_VEL
LIN {X 0,Y 421.299,Z 420.825,A -85,B 0,C 180,E1 18558.544,E2 18558.544} C_VEL
LIN {X 0,Y 416.853,Z 415.708,A -85,B 0,C 180,E1 18556.478,E2 18556.478} C_VEL
LIN {X 0,Y 415.772,Z 414.109,A -85,B 0,C 180,E1 18555.912,E2 18555.912} C_VEL
LIN {X 0,Y 412.366,Z 410.911,A -85,B 0,C 180,E1 18554.092,E2 18554.092} C_VEL
LIN {X 0,Y 410.586,Z 407.937,A -85,B 0,C 180,E1 18552.947,E2 18552.947} C_VEL
LIN {X 0,Y 407.105,Z 405.166,A -85,B 0,C 180,E1 18550.615,E2 18550.615} C_VEL
LIN {X 0,Y 405.262,Z 401.53,A -85,B 0,C 180,E1 18548.942,E2 18548.942} C_VEL
LIN {X 0,Y 401.47,Z 399.131,A -85,B 0,C 180,E1 18544.858,E2 18544.858} C_VEL
LIN {X 0,Y 399.74,Z 395.247,A -85,B 0,C 180,E1 18539.57,E2 18539.57} C_VEL
LIN {X 0,Y 399.742,Z 395.247,A -85,B 0,C 180,E1 18537.993,E2 18537.993} C_VEL
LIN {X 0,Y 401.877,Z 399.568,A -85,B 0,C 180,E1 18532.135,E2 18532.135} C_VEL
LIN {X 0,Y 405.347,Z 401.809,A -85,B 0,C 180,E1 18528.546,E2 18528.546} C_VEL
LIN {X 0,Y 407.325,Z 405.383,A -85,B 0,C 180,E1 18526.803,E2 18526.803} C_VEL
LIN {X 0,Y 410.405,Z 407.832,A -85,B 0,C 180,E1 18524.744,E2 18524.744} C_VEL
LIN {X 0,Y 411.097,Z 408.742,A -85,B 0,C 180,E1 18524.301,E2 18524.301} C_VEL
LIN {X 0,Y 413.993,Z 412.767,A -85,B 0,C 180,E1 18522.573,E2 18522.573} C_VEL
LIN {X 0,Y 416.281,Z 414.792,A -85,B 0,C 180,E1 18521.406,E2 18521.406} C_VEL
LIN {X 0,Y 419.453,Z 418.976,A -85,B 0,C 180,E1 18519.851,E2 18519.851} C_VEL
LIN {X 0,Y 421.308,Z 420.811,A -85,B 0,C 180,E1 18519.036,E2 18519.036} C_VEL
LIN {X 0,Y 425.07,Z 425.454,A -85,B 0,C 180,E1 18517.454,E2 18517.454} C_VEL
LIN {X 0,Y 427.658,Z 428.844,A -85,B 0,C 180,E1 18516.434,E2 18516.434} C_VEL
LIN {X 0,Y 431.094,Z 432.964,A -85,B 0,C 180,E1 18515.177,E2 18515.177} C_VEL
LIN {X 0,Y 435.975,Z 439.247,A -85,B 0,C 180,E1 18513.508,E2 18513.508} C_VEL
LIN {X 0,Y 442.658,Z 447.991,A -85,B 0,C 180,E1 18511.425,E2 18511.425} C_VEL
LIN {X 0,Y 452.49,Z 461.584,A -85,B 0,C 180,E1 18508.678,E2 18508.678} C_VEL
LIN {X 0,Y 462.744,Z 476.797,A -85,B 0,C 180,E1 18506.118,E2 18506.118} C_VEL
LIN {X 0,Y 472.652,Z 492.459,A -85,B 0,C 180,E1 18503.874,E2 18503.874} C_VEL
LIN {X 0,Y 458.666,Z 738.099,A -85,B 0,C 180,E1 18499.951,E2 18499.951} C_VEL
LIN {X 0,Y 456.752,Z 760.014,A -85,B 0,C 180,E1 18499.51,E2 18499.51} C_VEL
LIN {X 0,Y 453.479,Z 785.715,A -85,B 0,C 180,E1 18498.801,E2 18498.801} C_VEL
LIN {X 0,Y 450.166,Z 805.785,A -85,B 0,C 180,E1 18498.081,E2 18498.081} C_VEL
LIN {X 0,Y 445.801,Z 828.395,A -85,B 0,C 180,E1 18497.08,E2 18497.08} C_VEL
LIN {X 0,Y 440.536,Z 851.049,A -85,B 0,C 180,E1 18495.826,E2 18495.826} C_VEL
LIN {X 0,Y 435.215,Z 871.436,A -85,B 0,C 180,E1 18494.485,E2 18494.485} C_VEL
LIN {X 0,Y 428.993,Z 892.708,A -85,B 0,C 180,E1 18492.799,E2 18492.799} C_VEL
LIN {X 0,Y 423.304,Z 910.614,A -85,B 0,C 180,E1 18491.136,E2 18491.136} C_VEL
LIN {X 0,Y 416.422,Z 930.803,A -85,B 0,C 180,E1 18488.924,E2 18488.924} C_VEL
LIN {X 0,Y 410.742,Z 946.551,A -85,B 0,C 180,E1 18486.901,E2 18486.901} C_VEL
LIN {X 0,Y 404.223,Z 964.023,A -85,B 0,C 180,E1 18484.291,E2 18484.291} C_VEL
LIN {X 0,Y 398.77,Z 978.285,A -85,B 0,C 180,E1 18481.773,E2 18481.773} C_VEL
LIN {X 0,Y 393.418,Z 992.492,A -85,B 0,C 180,E1 18478.874,E2 18478.874} C_VEL
LIN {X 0,Y 388.636,Z 1005.189,A -85,B 0,C 180,E1 18475.773,E2 18475.773} C_VEL
LIN {X 0,Y 384.759,Z 1016.241,A -85,B 0,C 180,E1 18472.62,E2 18472.62} C_VEL
LIN {X 0,Y 381.461,Z 1026.344,A -85,B 0,C 180,E1 18469.126,E2 18469.126} C_VEL
LIN {X 0,Y 379.252,Z 1034.079,A -85,B 0,C 180,E1 18465.914,E2 18465.914} C_VEL
LIN {X 0,Y 377.506,Z 1041.462,A -85,B 0,C 180,E1 18462.078,E2 18462.078} C_VEL
LIN {X 0,Y 376.635,Z 1046.231,A -85,B 0,C 180,E1 18458.858,E2 18458.858} C_VEL
LIN {X 0,Y 376.175,Z 1050.124,A -85,B 0,C 180,E1 18455.338,E2 18455.338} C_VEL
LIN {X 0,Y 376.006,Z 1052.412,A -85,B 0,C 180,E1 18451.829,E2 18451.829} C_VEL
LIN {X 0,Y 375.97,Z 1053.298,A -85,B 0,C 180,E1 18448.933,E2 18448.933} C_VEL
LIN {X 0,Y 375.98,Z 1053.205,A -85,B 0,C 180,E1 18445.781,E2 18445.781} C_VEL
LIN {X 0,Y 376.077,Z 1051.718,A -85,B 0,C 180,E1 18442.207,E2 18442.207} C_VEL
LIN {X 0,Y 376.362,Z 1049.06,A -85,B 0,C 180,E1 18438.972,E2 18438.972} C_VEL
LIN {X 0,Y 376.991,Z 1045.229,A -85,B 0,C 180,E1 18435.72,E2 18435.72} C_VEL
LIN {X 0,Y 378.403,Z 1038.971,A -85,B 0,C 180,E1 18431.832,E2 18431.832} C_VEL
LIN {X 0,Y 380.312,Z 1032.182,A -85,B 0,C 180,E1 18428.547,E2 18428.547} C_VEL
LIN {X 0,Y 383.447,Z 1022.659,A -85,B 0,C 180,E1 18424.804,E2 18424.804} C_VEL
LIN {X 0,Y 384.449,Z 1019.742,A -85,B 0,C 180,E1 18423.812,E2 18423.812} C_VEL
LIN {X 0,Y 384.646,Z 1016.77,A -85,B 0,C 180,E1 18422.746,E2 18422.746} C_VEL
LIN {X 0,Y 382.131,Z 1008.67,A -85,B 0,C 180,E1 18419.834,E2 18419.834} C_VEL
LIN {X 0,Y 382.694,Z 1005.603,A -85,B 0,C 180,E1 18418.948,E2 18418.948} C_VEL
LIN {X 0,Y 388.256,Z 992.368,A -85,B 0,C 180,E1 18415.667,E2 18415.667} C_VEL
LIN {X 0,Y 394.017,Z 978.627,A -85,B 0,C 180,E1 18412.829,E2 18412.829} C_VEL
LIN {X 0,Y 400.549,Z 963.213,A -85,B 0,C 180,E1 18410.093,E2 18410.093} C_VEL
LIN {X 0,Y 407.452,Z 946.166,A -85,B 0,C 180,E1 18407.557,E2 18407.557} C_VEL
LIN {X 0,Y 414.186,Z 929.038,A -85,B 0,C 180,E1 18405.372,E2 18405.372} C_VEL
LIN {X 0,Y 421.151,Z 910.027,A -85,B 0,C 180,E1 18403.326,E2 18403.326} C_VEL
LIN {X 0,Y 427.212,Z 892.368,A -85,B 0,C 180,E1 18401.702,E2 18401.702} C_VEL
LIN {X 0,Y 434.282,Z 869.687,A -85,B 0,C 180,E1 18399.942,E2 18399.942} C_VEL
LIN {X 0,Y 439.772,Z 850.01,A -85,B 0,C 180,E1 18398.675,E2 18398.675} C_VEL
LIN {X 0,Y 445.565,Z 826.246,A -85,B 0,C 180,E1 18397.4,E2 18397.4} C_VEL
LIN {X 0,Y 449.848,Z 805.433,A -85,B 0,C 180,E1 18396.502,E2 18396.502} C_VEL
LIN {X 0,Y 453.959,Z 781.735,A -85,B 0,C 180,E1 18395.679,E2 18395.679} C_VEL
LIN {X 0,Y 457.039,Z 757.598,A -85,B 0,C 180,E1 18395.059,E2 18395.059} C_VEL
LIN {X 0,Y 459.217,Z 732.893,A -85,B 0,C 180,E1 18394.588,E2 18394.588} C_VEL
LIN {X 0,Y 473.455,Z 500.104,A -85,B 0,C 180,E1 18390.877,E2 18390.877} C_VEL
LIN {X 0,Y 463.328,Z 484.174,A -85,B 0,C 180,E1 18388.303,E2 18388.303} C_VEL
LIN {X 0,Y 453.867,Z 470.442,A -85,B 0,C 180,E1 18385.617,E2 18385.617} C_VEL
LIN {X 0,Y 446.179,Z 459.921,A -85,B 0,C 180,E1 18383.16,E2 18383.16} C_VEL
LIN {X 0,Y 439.936,Z 451.462,A -85,B 0,C 180,E1 18380.906,E2 18380.906} C_VEL
LIN {X 0,Y 435.12,Z 445.449,A -85,B 0,C 180,E1 18378.975,E2 18378.975} C_VEL
LIN {X 0,Y 431.297,Z 440.548,A -85,B 0,C 180,E1 18377.262,E2 18377.262} C_VEL
LIN {X 0,Y 427.805,Z 436.18,A -85,B 0,C 180,E1 18375.523,E2 18375.523} C_VEL
LIN {X 0,Y 426.589,Z 434.763,A -85,B 0,C 180,E1 18374.872,E2 18374.872} C_VEL
LIN {X 0,Y 423.245,Z 430.774,A -85,B 0,C 180,E1 18372.9,E2 18372.9} C_VEL
LIN {X 0,Y 422.373,Z 429.307,A -85,B 0,C 180,E1 18372.302,E2 18372.302} C_VEL
LIN {X 0,Y 418.943,Z 426.044,A -85,B 0,C 180,E1 18369.826,E2 18369.826} C_VEL
LIN {X 0,Y 417.474,Z 423.172,A -85,B 0,C 180,E1 18368.401,E2 18368.401} C_VEL
LIN {X 0,Y 413.613,Z 419.955,A -85,B 0,C 180,E1 18363.465,E2 18363.465} C_VEL
LIN {X 0,Y 412.773,Z 417.456,A -85,B 0,C 180,E1 18359.722,E2 18359.722} C_VEL
LIN {X 0,Y 412.842,Z 417.936,A -85,B 0,C 180,E1 18357.64,E2 18357.64} C_VEL
LIN {X 0,Y 417.027,Z 422.988,A -85,B 0,C 180,E1 18350.338,E2 18350.338} C_VEL
LIN {X 0,Y 417.682,Z 423.496,A -85,B 0,C 180,E1 18349.727,E2 18349.727} C_VEL
LIN {X 0,Y 419.856,Z 427.269,A -85,B 0,C 180,E1 18347.763,E2 18347.763} C_VEL
LIN {X 0,Y 422.682,Z 429.677,A -85,B 0,C 180,E1 18345.828,E2 18345.828} C_VEL
LIN {X 0,Y 425.518,Z 433.819,A -85,B 0,C 180,E1 18344.042,E2 18344.042} C_VEL
LIN {X 0,Y 427.645,Z 435.902,A -85,B 0,C 180,E1 18342.901,E2 18342.901} C_VEL
LIN {X 0,Y 431.324,Z 440.528,A -85,B 0,C 180,E1 18341.062,E2 18341.062} C_VEL
LIN {X 0,Y 437.04,Z 447.87,A -85,B 0,C 180,E1 18338.562,E2 18338.562} C_VEL
LIN {X 0,Y 442.601,Z 455.989,A -85,B 0,C 180,E1 18336.395,E2 18336.395} C_VEL
LIN {X 0,Y 449.951,Z 466.899,A -85,B 0,C 180,E1 18333.864,E2 18333.864} C_VEL
LIN {X 0,Y 459.467,Z 482.19,A -85,B 0,C 180,E1 18330.968,E2 18330.968} C_VEL
LIN {X 0,Y 468.305,Z 497.46,A -85,B 0,C 180,E1 18328.567,E2 18328.567} C_VEL
LIN {X 0,Y 473.26,Z 506.669,A -85,B 0,C 180,E1 18327.31,E2 18327.31} C_VEL
LIN {X 0,Y 458.128,Z 753.463,A -85,B 0,C 180,E1 18323.366,E2 18323.366} C_VEL
LIN {X 0,Y 455.966,Z 775.883,A -85,B 0,C 180,E1 18322.925,E2 18322.925} C_VEL
LIN {X 0,Y 452.132,Z 802.192,A -85,B 0,C 180,E1 18322.232,E2 18322.232} C_VEL
LIN {X 0,Y 448.34,Z 822.781,A -85,B 0,C 180,E1 18321.518,E2 18321.518} C_VEL
LIN {X 0,Y 443.19,Z 846.317,A -85,B 0,C 180,E1 18320.497,E2 18320.497} C_VEL
LIN {X 0,Y 437.935,Z 866.84,A -85,B 0,C 180,E1 18319.39,E2 18319.39} C_VEL
LIN {X 0,Y 432.081,Z 887.426,A -85,B 0,C 180,E1 18318.072,E2 18318.072} C_VEL
LIN {X 0,Y 425.546,Z 907.928,A -85,B 0,C 180,E1 18316.492,E2 18316.492} C_VEL
LIN {X 0,Y 419.209,Z 926.381,A -85,B 0,C 180,E1 18314.815,E2 18314.815} C_VEL
LIN {X 0,Y 411.637,Z 946.918,A -85,B 0,C 180,E1 18312.607,E2 18312.607} C_VEL
LIN {X 0,Y 405.349,Z 963.072,A -85,B 0,C 180,E1 18310.557,E2 18310.557} C_VEL
LIN {X 0,Y 398.317,Z 980.667,A -85,B 0,C 180,E1 18307.953,E2 18307.953} C_VEL
LIN {X 0,Y 392.19,Z 995.609,A -85,B 0,C 180,E1 18305.329,E2 18305.329} C_VEL
LIN {X 0,Y 386.377,Z 1010.038,A -85,B 0,C 180,E1 18302.391,E2 18302.391} C_VEL
LIN {X 0,Y 381.166,Z 1023.104,A -85,B 0,C 180,E1 18299.204,E2 18299.204} C_VEL
LIN {X 0,Y 376.92,Z 1034.573,A -85,B 0,C 180,E1 18295.934,E2 18295.934} C_VEL
LIN {X 0,Y 373.388,Z 1044.968,A -85,B 0,C 180,E1 18292.35,E2 18292.35} C_VEL
LIN {X 0,Y 371.048,Z 1053,A -85,B 0,C 180,E1 18289.03,E2 18289.03} C_VEL
LIN {X 0,Y 369.244,Z 1060.698,A -85,B 0,C 180,E1 18285.068,E2 18285.068} C_VEL
LIN {X 0,Y 368.41,Z 1065.687,A -85,B 0,C 180,E1 18281.745,E2 18281.745} C_VEL
LIN {X 0,Y 368.013,Z 1069.776,A -85,B 0,C 180,E1 18278.122,E2 18278.122} C_VEL
LIN {X 0,Y 367.949,Z 1072.2,A -85,B 0,C 180,E1 18274.52,E2 18274.52} C_VEL
LIN {X 0,Y 367.96,Z 1073.142,A -85,B 0,C 180,E1 18271.557,E2 18271.557} C_VEL
LIN {X 0,Y 367.964,Z 1073.092,A -85,B 0,C 180,E1 18268.599,E2 18268.599} C_VEL
LIN {X 0,Y 367.957,Z 1071.742,A -85,B 0,C 180,E1 18265.011,E2 18265.011} C_VEL
LIN {X 0,Y 368.049,Z 1068.787,A -85,B 0,C 180,E1 18261.454,E2 18261.454} C_VEL
LIN {X 0,Y 368.399,Z 1064.96,A -85,B 0,C 180,E1 18258.255,E2 18258.255} C_VEL
LIN {X 0,Y 369.37,Z 1058.884,A -85,B 0,C 180,E1 18254.455,E2 18254.455} C_VEL
LIN {X 0,Y 370.963,Z 1051.643,A -85,B 0,C 180,E1 18250.965,E2 18250.965} C_VEL
LIN {X 0,Y 373.52,Z 1042.506,A -85,B 0,C 180,E1 18247.327,E2 18247.327} C_VEL
LIN {X 0,Y 376.915,Z 1031.81,A -85,B 0,C 180,E1 18243.873,E2 18243.873} C_VEL
LIN {X 0,Y 381.193,Z 1019.77,A -85,B 0,C 180,E1 18240.559,E2 18240.559} C_VEL
LIN {X 0,Y 386.259,Z 1006.087,A -85,B 0,C 180,E1 18237.423,E2 18237.423} C_VEL
LIN {X 0,Y 391.772,Z 991.744,A -85,B 0,C 180,E1 18234.595,E2 18234.595} C_VEL
LIN {X 0,Y 398.151,Z 975.046,A -85,B 0,C 180,E1 18231.818,E2 18231.818} C_VEL
LIN {X 0,Y 404.06,Z 959.404,A -85,B 0,C 180,E1 18229.583,E2 18229.583} C_VEL
LIN {X 0,Y 411.225,Z 939.668,A -85,B 0,C 180,E1 18227.188,E2 18227.188} C_VEL
LIN {X 0,Y 417.284,Z 922.041,A -85,B 0,C 180,E1 18225.371,E2 18225.371} C_VEL
LIN {X 0,Y 424.273,Z 900.17,A -85,B 0,C 180,E1 18223.459,E2 18223.459} C_VEL
LIN {X 0,Y 429.916,Z 880.895,A -85,B 0,C 180,E1 18222.054,E2 18222.054} C_VEL
LIN {X 0,Y 435.801,Z 858.702,A -85,B 0,C 180,E1 18220.686,E2 18220.686} C_VEL
LIN {X 0,Y 440.76,Z 836.985,A -85,B 0,C 180,E1 18219.603,E2 18219.603} C_VEL
LIN {X 0,Y 444.917,Z 816.254,A -85,B 0,C 180,E1 18218.755,E2 18218.755} C_VEL
LIN {X 0,Y 449.001,Z 791.127,A -85,B 0,C 180,E1 18217.955,E2 18217.955} C_VEL
LIN {X 0,Y 451.686,Z 769.398,A -85,B 0,C 180,E1 18217.431,E2 18217.431} C_VEL
LIN {X 0,Y 454.073,Z 736.841,A -85,B 0,C 180,E1 18216.847,E2 18216.847} C_VEL
LIN {X 0,Y 467.644,Z 503.033,A -85,B 0,C 180,E1 18213.101,E2 18213.101} C_VEL
LIN {X 0,Y 457.829,Z 485.159,A -85,B 0,C 180,E1 18210.734,E2 18210.734} C_VEL
LIN {X 0,Y 448.434,Z 469.378,A -85,B 0,C 180,E1 18208.246,E2 18208.246} C_VEL
LIN {X 0,Y 439.686,Z 455.676,A -85,B 0,C 180,E1 18205.672,E2 18205.672} C_VEL
LIN {X 0,Y 431.475,Z 443.557,A -85,B 0,C 180,E1 18202.948,E2 18202.948} C_VEL
LIN {X 0,Y 427.074,Z 437.891,A -85,B 0,C 180,E1 18201.35,E2 18201.35} C_VEL
LIN {X 0,Y 423.034,Z 432.801,A -85,B 0,C 180,E1 18199.755,E2 18199.755} C_VEL
LIN {X 0,Y 419.299,Z 427.956,A -85,B 0,C 180,E1 18198.132,E2 18198.132} C_VEL
LIN {X 0,Y 415.399,Z 423.561,A -85,B 0,C 180,E1 18196.285,E2 18196.285} C_VEL
LIN {X 0,Y 414.009,Z 421.639,A -85,B 0,C 180,E1 18195.55,E2 18195.55} C_VEL
LIN {X 0,Y 410.724,Z 418.316,A -85,B 0,C 180,E1 18193.731,E2 18193.731} C_VEL
LIN {X 0,Y 409.172,Z 415.703,A -85,B 0,C 180,E1 18192.705,E2 18192.705} C_VEL
LIN {X 0,Y 405.686,Z 412.733,A -85,B 0,C 180,E1 18190.293,E2 18190.293} C_VEL
LIN {X 0,Y 403.962,Z 409.372,A -85,B 0,C 180,E1 18188.684,E2 18188.684} C_VEL
LIN {X 0,Y 400.228,Z 406.777,A -85,B 0,C 180,E1 18184.442,E2 18184.442} C_VEL
LIN {X 0,Y 398.765,Z 403.19,A -85,B 0,C 180,E1 18179.569,E2 18179.569} C_VEL
LIN {X 0,Y 398.764,Z 403.218,A -85,B 0,C 180,E1 18177.988,E2 18177.988} C_VEL
LIN {X 0,Y 402.905,Z 408.947,A -85,B 0,C 180,E1 18169.851,E2 18169.851} C_VEL
LIN {X 0,Y 404.064,Z 409.552,A -85,B 0,C 180,E1 18168.799,E2 18168.799} C_VEL
LIN {X 0,Y 406.171,Z 413.304,A -85,B 0,C 180,E1 18166.91,E2 18166.91} C_VEL
LIN {X 0,Y 409.485,Z 416.11,A -85,B 0,C 180,E1 18164.673,E2 18164.673} C_VEL
LIN {X 0,Y 412.414,Z 420.34,A -85,B 0,C 180,E1 18162.868,E2 18162.868} C_VEL
LIN {X 0,Y 414.717,Z 422.496,A -85,B 0,C 180,E1 18161.661,E2 18161.661} C_VEL
LIN {X 0,Y 418.065,Z 426.807,A -85,B 0,C 180,E1 18160,E2 18160} C_VEL
LIN {X 0,Y 419.667,Z 428.537,A -85,B 0,C 180,E1 18159.279,E2 18159.279} C_VEL
LIN {X 0,Y 423.636,Z 433.301,A -85,B 0,C 180,E1 18157.593,E2 18157.593} C_VEL
LIN {X 0,Y 429.418,Z 440.849,A -85,B 0,C 180,E1 18155.367,E2 18155.367} C_VEL
LIN {X 0,Y 434.165,Z 447.01,A -85,B 0,C 180,E1 18153.72,E2 18153.72} C_VEL
LIN {X 0,Y 440.974,Z 456.175,A -85,B 0,C 180,E1 18151.564,E2 18151.564} C_VEL
LIN {X 0,Y 449.772,Z 468.497,A -85,B 0,C 180,E1 18149.063,E2 18149.063} C_VEL
LIN {X 0,Y 459.776,Z 483.553,A -85,B 0,C 180,E1 18146.507,E2 18146.507} C_VEL
LIN {X 0,Y 467.865,Z 496.717,A -85,B 0,C 180,E1 18144.611,E2 18144.611} C_VEL
LIN {X 0,Y 453.549,Z 740.077,A -85,B 0,C 180,E1 18140.706,E2 18140.706} C_VEL
LIN {X 0,Y 451.468,Z 762.645,A -85,B 0,C 180,E1 18140.24,E2 18140.24} C_VEL
LIN {X 0,Y 448.099,Z 787.565,A -85,B 0,C 180,E1 18139.531,E2 18139.531} C_VEL
LIN {X 0,Y 444.73,Z 807.284,A -85,B 0,C 180,E1 18138.812,E2 18138.812} C_VEL
LIN {X 0,Y 439.958,Z 830.893,A -85,B 0,C 180,E1 18137.742,E2 18137.742} C_VEL
LIN {X 0,Y 434.991,Z 851.578,A -85,B 0,C 180,E1 18136.583,E2 18136.583} C_VEL
LIN {X 0,Y 429.294,Z 872.789,A -85,B 0,C 180,E1 18135.176,E2 18135.176} C_VEL
LIN {X 0,Y 423.117,Z 893.156,A -85,B 0,C 180,E1 18133.54,E2 18133.54} C_VEL
LIN {X 0,Y 417.04,Z 911.701,A -85,B 0,C 180,E1 18131.8,E2 18131.8} C_VEL
LIN {X 0,Y 410.018,Z 931.561,A -85,B 0,C 180,E1 18129.591,E2 18129.591} C_VEL
LIN {X 0,Y 404.138,Z 947.318,A -85,B 0,C 180,E1 18127.538,E2 18127.538} C_VEL
LIN {X 0,Y 397.273,Z 965.01,A -85,B 0,C 180,E1 18124.843,E2 18124.843} C_VEL
LIN {X 0,Y 391.57,Z 979.385,A -85,B 0,C 180,E1 18122.255,E2 18122.255} C_VEL
LIN {X 0,Y 385.699,Z 994.267,A -85,B 0,C 180,E1 18119.115,E2 18119.115} C_VEL
LIN {X 0,Y 381.095,Z 1006.064,A -85,B 0,C 180,E1 18116.154,E2 18116.154} C_VEL
LIN {X 0,Y 376.909,Z 1017.523,A -85,B 0,C 180,E1 18112.788,E2 18112.788} C_VEL
LIN {X 0,Y 373.528,Z 1027.42,A -85,B 0,C 180,E1 18109.224,E2 18109.224} C_VEL
LIN {X 0,Y 371.105,Z 1035.73,A -85,B 0,C 180,E1 18105.631,E2 18105.631} C_VEL
LIN {X 0,Y 369.496,Z 1042.216,A -85,B 0,C 180,E1 18102.027,E2 18102.027} C_VEL
LIN {X 0,Y 368.621,Z 1046.883,A -85,B 0,C 180,E1 18098.737,E2 18098.737} C_VEL
LIN {X 0,Y 368.137,Z 1050.811,A -85,B 0,C 180,E1 18094.83,E2 18094.83} C_VEL
LIN {X 0,Y 368.003,Z 1052.77,A -85,B 0,C 180,E1 18091.557,E2 18091.557} C_VEL
LIN {X 0,Y 367.963,Z 1053.583,A -85,B 0,C 180,E1 18088.443,E2 18088.443} C_VEL
LIN {X 0,Y 367.998,Z 1053.234,A -85,B 0,C 180,E1 18084.856,E2 18084.856} C_VEL
LIN {X 0,Y 368.14,Z 1051.47,A -85,B 0,C 180,E1 18081.409,E2 18081.409} C_VEL
LIN {X 0,Y 368.47,Z 1048.781,A -85,B 0,C 180,E1 18078.257,E2 18078.257} C_VEL
LIN {X 0,Y 369.381,Z 1044.115,A -85,B 0,C 180,E1 18074.455,E2 18074.455} C_VEL
LIN {X 0,Y 370.849,Z 1038.244,A -85,B 0,C 180,E1 18070.959,E2 18070.959} C_VEL
LIN {X 0,Y 373.227,Z 1030.64,A -85,B 0,C 180,E1 18067.308,E2 18067.308} C_VEL
LIN {X 0,Y 376.569,Z 1021.105,A -85,B 0,C 180,E1 18063.677,E2 18063.677} C_VEL
LIN {X 0,Y 380.596,Z 1010.851,A -85,B 0,C 180,E1 18060.402,E2 18060.402} C_VEL
LIN {X 0,Y 382.694,Z 1005.603,A -85,B 0,C 180,E1 18058.948,E2 18058.948} C_VEL
LIN {X 0,Y 383.317,Z 1002.103,A -85,B 0,C 180,E1 18057.919,E2 18057.919} C_VEL
LIN {X 0,Y 381.972,Z 992.669,A -85,B 0,C 180,E1 18055.075,E2 18055.075} C_VEL
LIN {X 0,Y 382.854,Z 989.136,A -85,B 0,C 180,E1 18054.234,E2 18054.234} C_VEL
LIN {X 0,Y 388.792,Z 975.723,A -85,B 0,C 180,E1 18051.51,E2 18051.51} C_VEL
LIN {X 0,Y 395.749,Z 959.633,A -85,B 0,C 180,E1 18048.743,E2 18048.743} C_VEL
LIN {X 0,Y 402.235,Z 944.199,A -85,B 0,C 180,E1 18046.482,E2 18046.482} C_VEL
LIN {X 0,Y 409.965,Z 924.952,A -85,B 0,C 180,E1 18044.088,E2 18044.088} C_VEL
LIN {X 0,Y 416.614,Z 907.166,A -85,B 0,C 180,E1 18042.223,E2 18042.223} C_VEL
LIN {X 0,Y 423.872,Z 886.302,A -85,B 0,C 180,E1 18040.365,E2 18040.365} C_VEL
LIN {X 0,Y 429.927,Z 866.82,A -85,B 0,C 180,E1 18038.916,E2 18038.916} C_VEL
LIN {X 0,Y 436.219,Z 844.593,A -85,B 0,C 180,E1 18037.525,E2 18037.525} C_VEL
LIN {X 0,Y 441.487,Z 822.45,A -85,B 0,C 180,E1 18036.398,E2 18036.398} C_VEL
LIN {X 0,Y 445.876,Z 801.155,A -85,B 0,C 180,E1 18035.508,E2 18035.508} C_VEL
LIN {X 0,Y 449.985,Z 776.229,A -85,B 0,C 180,E1 18034.699,E2 18034.699} C_VEL
LIN {X 0,Y 452.779,Z 754.059,A -85,B 0,C 180,E1 18034.157,E2 18034.157} C_VEL
LIN {X 0,Y 455.317,Z 721.258,A -85,B 0,C 180,E1 18033.578,E2 18033.578} C_VEL
LIN {X 0,Y 469.023,Z 504.436,A -85,B 0,C 180,E1 18030.119,E2 18030.119} C_VEL
LIN {X 0,Y 459.73,Z 489.717,A -85,B 0,C 180,E1 18027.668,E2 18027.668} C_VEL
LIN {X 0,Y 451.14,Z 477.063,A -85,B 0,C 180,E1 18025.15,E2 18025.15} C_VEL
LIN {X 0,Y 443.696,Z 466.703,A -85,B 0,C 180,E1 18022.701,E2 18022.701} C_VEL
LIN {X 0,Y 437.661,Z 458.472,A -85,B 0,C 180,E1 18020.46,E2 18020.46} C_VEL
LIN {X 0,Y 433.252,Z 452.826,A -85,B 0,C 180,E1 18018.641,E2 18018.641} C_VEL
LIN {X 0,Y 429.5,Z 447.972,A -85,B 0,C 180,E1 18016.918,E2 18016.918} C_VEL
LIN {X 0,Y 425.925,Z 443.233,A -85,B 0,C 180,E1 18015.07,E2 18015.07} C_VEL
LIN {X 0,Y 421.947,Z 438.647,A -85,B 0,C 180,E1 18012.732,E2 18012.732} C_VEL
LIN {X 0,Y 420.99,Z 437.062,A -85,B 0,C 180,E1 18012.064,E2 18012.064} C_VEL
LIN {X 0,Y 417.57,Z 433.613,A -85,B 0,C 180,E1 18009.51,E2 18009.51} C_VEL
LIN {X 0,Y 416.205,Z 431.007,A -85,B 0,C 180,E1 18008.149,E2 18008.149} C_VEL
LIN {X 0,Y 412.17,Z 427.007,A -85,B 0,C 180,E1 18002.225,E2 18002.225} C_VEL
LIN {X 0,Y 411.795,Z 425.299,A -85,B 0,C 180,E1 17999.444,E2 17999.444} C_VEL
LIN {X 0,Y 411.898,Z 426.108,A -85,B 0,C 180,E1 17997.356,E2 17997.356} C_VEL
LIN {X 0,Y 415.919,Z 430.884,A -85,B 0,C 180,E1 17990.452,E2 17990.452} C_VEL
LIN {X 0,Y 416.55,Z 431.513,A -85,B 0,C 180,E1 17989.838,E2 17989.838} C_VEL
LIN {X 0,Y 418.885,Z 435.355,A -85,B 0,C 180,E1 17987.734,E2 17987.734} C_VEL
LIN {X 0,Y 421.301,Z 437.421,A -85,B 0,C 180,E1 17986.061,E2 17986.061} C_VEL
LIN {X 0,Y 424.321,Z 441.746,A -85,B 0,C 180,E1 17984.136,E2 17984.136} C_VEL
LIN {X 0,Y 426.118,Z 443.564,A -85,B 0,C 180,E1 17983.154,E2 17983.154} C_VEL
LIN {X 0,Y 429.95,Z 448.349,A -85,B 0,C 180,E1 17981.21,E2 17981.21} C_VEL
LIN {X 0,Y 435.295,Z 455.466,A -85,B 0,C 180,E1 17978.825,E2 17978.825} C_VEL
LIN {X 0,Y 440.693,Z 463.515,A -85,B 0,C 180,E1 17976.676,E2 17976.676} C_VEL
LIN {X 0,Y 447.764,Z 474.27,A -85,B 0,C 180,E1 17974.186,E2 17974.186} C_VEL
LIN {X 0,Y 456.781,Z 488.986,A -85,B 0,C 180,E1 17971.376,E2 17971.376} C_VEL
LIN {X 0,Y 465.329,Z 504.068,A -85,B 0,C 180,E1 17968.991,E2 17968.991} C_VEL
LIN {X 0,Y 468.796,Z 510.797,A -85,B 0,C 180,E1 17968.077,E2 17968.077} C_VEL
LIN {X 0,Y 453.357,Z 754.88,A -85,B 0,C 180,E1 17964.161,E2 17964.161} C_VEL
LIN {X 0,Y 450.926,Z 778.675,A -85,B 0,C 180,E1 17963.684,E2 17963.684} C_VEL
LIN {X 0,Y 447.1,Z 803.382,A -85,B 0,C 180,E1 17963.014,E2 17963.014} C_VEL
LIN {X 0,Y 443.092,Z 824.425,A -85,B 0,C 180,E1 17962.274,E2 17962.274} C_VEL
LIN {X 0,Y 437.526,Z 848.652,A -85,B 0,C 180,E1 17961.196,E2 17961.196} C_VEL
LIN {X 0,Y 432.44,Z 867.888,A -85,B 0,C 180,E1 17960.143,E2 17960.143} C_VEL
LIN {X 0,Y 425.904,Z 890.012,A -85,B 0,C 180,E1 17958.7,E2 17958.7} C_VEL
LIN {X 0,Y 419.385,Z 909.625,A -85,B 0,C 180,E1 17957.15,E2 17957.15} C_VEL
LIN {X 0,Y 412.739,Z 928.342,A -85,B 0,C 180,E1 17955.417,E2 17955.417} C_VEL
LIN {X 0,Y 405.103,Z 948.175,A -85,B 0,C 180,E1 17953.231,E2 17953.231} C_VEL
LIN {X 0,Y 398.482,Z 964.6,A -85,B 0,C 180,E1 17951.104,E2 17951.104} C_VEL
LIN {X 0,Y 391.099,Z 982.254,A -85,B 0,C 180,E1 17948.408,E2 17948.408} C_VEL
LIN {X 0,Y 385.189,Z 996.151,A -85,B 0,C 180,E1 17945.913,E2 17945.913} C_VEL
LIN {X 0,Y 378.842,Z 1011.201,A -85,B 0,C 180,E1 17942.756,E2 17942.756} C_VEL
LIN {X 0,Y 373.719,Z 1023.535,A -85,B 0,C 180,E1 17939.668,E2 17939.668} C_VEL
LIN {X 0,Y 369.151,Z 1035.366,A -85,B 0,C 180,E1 17936.2,E2 17936.2} C_VEL
LIN {X 0,Y 365.626,Z 1045.209,A -85,B 0,C 180,E1 17932.681,E2 17932.681} C_VEL
LIN {X 0,Y 363.088,Z 1053.541,A -85,B 0,C 180,E1 17929.13,E2 17929.13} C_VEL
LIN {X 0,Y 361.296,Z 1060.77,A -85,B 0,C 180,E1 17925.243,E2 17925.243} C_VEL
LIN {X 0,Y 360.425,Z 1065.706,A -85,B 0,C 180,E1 17921.847,E2 17921.847} C_VEL
LIN {X 0,Y 360.004,Z 1069.826,A -85,B 0,C 180,E1 17917.983,E2 17917.983} C_VEL
LIN {X 0,Y 359.952,Z 1071.994,A -85,B 0,C 180,E1 17914.621,E2 17914.621} C_VEL
LIN {X 0,Y 359.962,Z 1072.932,A -85,B 0,C 180,E1 17911.592,E2 17911.592} C_VEL
LIN {X 0,Y 359.966,Z 1072.875,A -85,B 0,C 180,E1 17908.568,E2 17908.568} C_VEL
LIN {X 0,Y 359.958,Z 1071.612,A -85,B 0,C 180,E1 17905.06,E2 17905.06} C_VEL
LIN {X 0,Y 360.053,Z 1068.647,A -85,B 0,C 180,E1 17901.356,E2 17901.356} C_VEL
LIN {X 0,Y 360.413,Z 1064.93,A -85,B 0,C 180,E1 17898.153,E2 17898.153} C_VEL
LIN {X 0,Y 361.408,Z 1059.041,A -85,B 0,C 180,E1 17894.323,E2 17894.323} C_VEL
LIN {X 0,Y 363.091,Z 1051.74,A -85,B 0,C 180,E1 17890.703,E2 17890.703} C_VEL
LIN {X 0,Y 365.622,Z 1043.077,A -85,B 0,C 180,E1 17887.149,E2 17887.149} C_VEL
LIN {X 0,Y 369.3,Z 1032.048,A -85,B 0,C 180,E1 17883.465,E2 17883.465} C_VEL
LIN {X 0,Y 373.422,Z 1020.87,A -85,B 0,C 180,E1 17880.306,E2 17880.306} C_VEL
LIN {X 0,Y 379.003,Z 1006.487,A -85,B 0,C 180,E1 17876.9,E2 17876.9} C_VEL
LIN {X 0,Y 384.385,Z 992.988,A -85,B 0,C 180,E1 17874.177,E2 17874.177} C_VEL
LIN {X 0,Y 391.357,Z 975.51,A -85,B 0,C 180,E1 17871.193,E2 17871.193} C_VEL
LIN {X 0,Y 397.396,Z 960.08,A -85,B 0,C 180,E1 17868.951,E2 17868.951} C_VEL
LIN {X 0,Y 404.992,Z 939.906,A -85,B 0,C 180,E1 17866.463,E2 17866.463} C_VEL
LIN {X 0,Y 411.158,Z 922.544,A -85,B 0,C 180,E1 17864.654,E2 17864.654} C_VEL
LIN {X 0,Y 418.181,Z 901.381,A -85,B 0,C 180,E1 17862.773,E2 17862.773} C_VEL
LIN {X 0,Y 424.222,Z 881.357,A -85,B 0,C 180,E1 17861.297,E2 17861.297} C_VEL
LIN {X 0,Y 430.263,Z 859.322,A -85,B 0,C 180,E1 17859.925,E2 17859.925} C_VEL
LIN {X 0,Y 435.549,Z 836.78,A -85,B 0,C 180,E1 17858.795,E2 17858.795} C_VEL
LIN {X 0,Y 439.892,Z 815.654,A -85,B 0,C 180,E1 17857.932,E2 17857.932} C_VEL
LIN {X 0,Y 444.031,Z 790.684,A -85,B 0,C 180,E1 17857.141,E2 17857.141} C_VEL
LIN {X 0,Y 446.787,Z 768.832,A -85,B 0,C 180,E1 17856.616,E2 17856.616} C_VEL
LIN {X 0,Y 449.223,Z 736.198,A -85,B 0,C 180,E1 17856.031,E2 17856.031} C_VEL
LIN {X 0,Y 462.936,Z 506.836,A -85,B 0,C 180,E1 17852.339,E2 17852.339} C_VEL
LIN {X 0,Y 453.675,Z 489.843,A -85,B 0,C 180,E1 17850.02,E2 17850.02} C_VEL
LIN {X 0,Y 445.019,Z 475.093,A -85,B 0,C 180,E1 17847.644,E2 17847.644} C_VEL
LIN {X 0,Y 436.749,Z 462.007,A -85,B 0,C 180,E1 17845.131,E2 17845.131} C_VEL
LIN {X 0,Y 429.076,Z 450.432,A -85,B 0,C 180,E1 17842.505,E2 17842.505} C_VEL
LIN {X 0,Y 424.757,Z 444.874,A -85,B 0,C 180,E1 17840.894,E2 17840.894} C_VEL
LIN {X 0,Y 421.117,Z 440.183,A -85,B 0,C 180,E1 17839.415,E2 17839.415} C_VEL
LIN {X 0,Y 416.87,Z 434.813,A -85,B 0,C 180,E1 17837.519,E2 17837.519} C_VEL
LIN {X 0,Y 413.273,Z 430.311,A -85,B 0,C 180,E1 17835.723,E2 17835.723} C_VEL
LIN {X 0,Y 412.265,Z 429.153,A -85,B 0,C 180,E1 17835.185,E2 17835.185} C_VEL
LIN {X 0,Y 408.976,Z 425.523,A -85,B 0,C 180,E1 17833.286,E2 17833.286} C_VEL
LIN {X 0,Y 407.766,Z 423.461,A -85,B 0,C 180,E1 17832.462,E2 17832.462} C_VEL
LIN {X 0,Y 404.364,Z 420.418,A -85,B 0,C 180,E1 17830.04,E2 17830.04} C_VEL
LIN {X 0,Y 402.672,Z 417.207,A -85,B 0,C 180,E1 17828.424,E2 17828.424} C_VEL
LIN {X 0,Y 399.086,Z 414.532,A -85,B 0,C 180,E1 17824.167,E2 17824.167} C_VEL
LIN {X 0,Y 397.781,Z 411.103,A -85,B 0,C 180,E1 17819.424,E2 17819.424} C_VEL
LIN {X 0,Y 397.785,Z 411.188,A -85,B 0,C 180,E1 17817.983,E2 17817.983} C_VEL
LIN {X 0,Y 401.797,Z 416.836,A -85,B 0,C 180,E1 17809.968,E2 17809.968} C_VEL
LIN {X 0,Y 402.918,Z 417.633,A -85,B 0,C 180,E1 17808.911,E2 17808.911} C_VEL
LIN {X 0,Y 405.199,Z 421.43,A -85,B 0,C 180,E1 17806.878,E2 17806.878} C_VEL
LIN {X 0,Y 408.13,Z 423.971,A -85,B 0,C 180,E1 17804.875,E2 17804.875} C_VEL
LIN {X 0,Y 411.209,Z 428.274,A -85,B 0,C 180,E1 17802.962,E2 17802.962} C_VEL
LIN {X 0,Y 413.164,Z 430.186,A -85,B 0,C 180,E1 17801.918,E2 17801.918} C_VEL
LIN {X 0,Y 416.681,Z 434.634,A -85,B 0,C 180,E1 17800.15,E2 17800.15} C_VEL
LIN {X 0,Y 418.245,Z 436.571,A -85,B 0,C 180,E1 17799.425,E2 17799.425} C_VEL
LIN {X 0,Y 422.722,Z 442.153,A -85,B 0,C 180,E1 17797.505,E2 17797.505} C_VEL
LIN {X 0,Y 427.325,Z 448.118,A -85,B 0,C 180,E1 17795.717,E2 17795.717} C_VEL
LIN {X 0,Y 433.757,Z 456.516,A -85,B 0,C 180,E1 17793.472,E2 17793.472} C_VEL
LIN {X 0,Y 443.951,Z 470.767,A -85,B 0,C 180,E1 17790.335,E2 17790.335} C_VEL
LIN {X 0,Y 453.574,Z 485.262,A -85,B 0,C 180,E1 17787.721,E2 17787.721} C_VEL
LIN {X 0,Y 463.165,Z 500.599,A -85,B 0,C 180,E1 17785.373,E2 17785.373} C_VEL
LIN {X 0,Y 448.659,Z 740.144,A -85,B 0,C 180,E1 17781.511,E2 17781.511} C_VEL
LIN {X 0,Y 446.546,Z 762.536,A -85,B 0,C 180,E1 17781.049,E2 17781.049} C_VEL
LIN {X 0,Y 443.089,Z 787.592,A -85,B 0,C 180,E1 17780.339,E2 17780.339} C_VEL
LIN {X 0,Y 439.523,Z 807.94,A -85,B 0,C 180,E1 17779.595,E2 17779.595} C_VEL
LIN {X 0,Y 434.441,Z 832.213,A -85,B 0,C 180,E1 17778.482,E2 17778.482} C_VEL
LIN {X 0,Y 429.506,Z 852.174,A -85,B 0,C 180,E1 17777.355,E2 17777.355} C_VEL
LIN {X 0,Y 423.414,Z 874.165,A -85,B 0,C 180,E1 17775.881,E2 17775.881} C_VEL
LIN {X 0,Y 417.077,Z 894.328,A -85,B 0,C 180,E1 17774.238,E2 17774.238} C_VEL
LIN {X 0,Y 410.614,Z 913.446,A -85,B 0,C 180,E1 17772.417,E2 17772.417} C_VEL
LIN {X 0,Y 403.671,Z 932.318,A -85,B 0,C 180,E1 17770.278,E2 17770.278} C_VEL
LIN {X 0,Y 397.633,Z 947.961,A -85,B 0,C 180,E1 17768.213,E2 17768.213} C_VEL
LIN {X 0,Y 390.277,Z 966.194,A -85,B 0,C 180,E1 17765.381,E2 17765.381} C_VEL
LIN {X 0,Y 384.706,Z 979.727,A -85,B 0,C 180,E1 17762.903,E2 17762.903} C_VEL
LIN {X 0,Y 378.679,Z 994.392,A -85,B 0,C 180,E1 17759.763,E2 17759.763} C_VEL
LIN {X 0,Y 373.754,Z 1006.473,A -85,B 0,C 180,E1 17756.678,E2 17756.678} C_VEL
LIN {X 0,Y 369.412,Z 1017.815,A -85,B 0,C 180,E1 17753.277,E2 17753.277} C_VEL
LIN {X 0,Y 365.987,Z 1027.307,A -85,B 0,C 180,E1 17749.802,E2 17749.802} C_VEL
LIN {X 0,Y 363.389,Z 1035.666,A -85,B 0,C 180,E1 17746.135,E2 17746.135} C_VEL
LIN {X 0,Y 361.597,Z 1042.474,A -85,B 0,C 180,E1 17742.294,E2 17742.294} C_VEL
LIN {X 0,Y 360.667,Z 1047.132,A -85,B 0,C 180,E1 17738.931,E2 17738.931} C_VEL
LIN {X 0,Y 360.15,Z 1051.044,A -85,B 0,C 180,E1 17734.937,E2 17734.937} C_VEL
LIN {X 0,Y 360.011,Z 1052.928,A -85,B 0,C 180,E1 17731.751,E2 17731.751} C_VEL
LIN {X 0,Y 359.971,Z 1053.755,A -85,B 0,C 180,E1 17728.727,E2 17728.727} C_VEL
LIN {X 0,Y 359.993,Z 1053.576,A -85,B 0,C 180,E1 17725.22,E2 17725.22} C_VEL
LIN {X 0,Y 360.142,Z 1051.888,A -85,B 0,C 180,E1 17721.538,E2 17721.538} C_VEL
LIN {X 0,Y 360.474,Z 1049.252,A -85,B 0,C 180,E1 17718.284,E2 17718.284} C_VEL
LIN {X 0,Y 361.347,Z 1044.99,A -85,B 0,C 180,E1 17714.595,E2 17714.595} C_VEL
LIN {X 0,Y 362.996,Z 1038.712,A -85,B 0,C 180,E1 17710.698,E2 17710.698} C_VEL
LIN {X 0,Y 365.225,Z 1031.847,A -85,B 0,C 180,E1 17707.293,E2 17707.293} C_VEL
LIN {X 0,Y 368.807,Z 1022.158,A -85,B 0,C 180,E1 17703.427,E2 17703.427} C_VEL
LIN {X 0,Y 372.735,Z 1012.517,A -85,B 0,C 180,E1 17700.246,E2 17700.246} C_VEL
LIN {X 0,Y 378.376,Z 999.354,A -85,B 0,C 180,E1 17696.622,E2 17696.622} C_VEL
LIN {X 0,Y 382.854,Z 989.136,A -85,B 0,C 180,E1 17694.234,E2 17694.234} C_VEL
LIN {X 0,Y 383.853,Z 985.086,A -85,B 0,C 180,E1 17693.26,E2 17693.26} C_VEL
LIN {X 0,Y 383.625,Z 974.33,A -85,B 0,C 180,E1 17690.522,E2 17690.522} C_VEL
LIN {X 0,Y 384.786,Z 970.371,A -85,B 0,C 180,E1 17689.74,E2 17689.74} C_VEL
LIN {X 0,Y 391.207,Z 956.01,A -85,B 0,C 180,E1 17687.366,E2 17687.366} C_VEL
LIN {X 0,Y 398.981,Z 937.989,A -85,B 0,C 180,E1 17684.828,E2 17684.828} C_VEL
LIN {X 0,Y 405.645,Z 921.531,A -85,B 0,C 180,E1 17682.869,E2 17682.869} C_VEL
LIN {X 0,Y 412.922,Z 902.567,A -85,B 0,C 180,E1 17680.93,E2 17680.93} C_VEL
LIN {X 0,Y 419.945,Z 882.198,A -85,B 0,C 180,E1 17679.193,E2 17679.193} C_VEL
LIN {X 0,Y 425.953,Z 863.235,A -85,B 0,C 180,E1 17677.823,E2 17677.823} C_VEL
LIN {X 0,Y 432.451,Z 839.933,A -85,B 0,C 180,E1 17676.426,E2 17676.426} C_VEL
LIN {X 0,Y 437.087,Z 820.715,A -85,B 0,C 180,E1 17675.473,E2 17675.473} C_VEL
LIN {X 0,Y 441.996,Z 796.971,A -85,B 0,C 180,E1 17674.512,E2 17674.512} C_VEL
LIN {X 0,Y 445.667,Z 774.241,A -85,B 0,C 180,E1 17673.803,E2 17673.803} C_VEL
LIN {X 0,Y 448.734,Z 749.707,A -85,B 0,C 180,E1 17673.225,E2 17673.225} C_VEL
LIN {X 0,Y 452.235,Z 698.908,A -85,B 0,C 180,E1 17672.378,E2 17672.378} C_VEL
LIN {X 0,Y 464.59,Z 508.604,A -85,B 0,C 180,E1 17669.323,E2 17669.323} C_VEL
LIN {X 0,Y 455.479,Z 494.085,A -85,B 0,C 180,E1 17666.816,E2 17666.816} C_VEL
LIN {X 0,Y 446.434,Z 480.677,A -85,B 0,C 180,E1 17664.021,E2 17664.021} C_VEL
LIN {X 0,Y 438.584,Z 469.793,A -85,B 0,C 180,E1 17661.253,E2 17661.253} C_VEL
LIN {X 0,Y 434.792,Z 464.712,A -85,B 0,C 180,E1 17659.759,E2 17659.759} C_VEL
LIN {X 0,Y 431.544,Z 460.364,A -85,B 0,C 180,E1 17658.368,E2 17658.368} C_VEL
LIN {X 0,Y 427.72,Z 455.387,A -85,B 0,C 180,E1 17656.571,E2 17656.571} C_VEL
LIN {X 0,Y 423.811,Z 450.255,A -85,B 0,C 180,E1 17654.483,E2 17654.483} C_VEL
LIN {X 0,Y 420.368,Z 446.019,A -85,B 0,C 180,E1 17652.361,E2 17652.361} C_VEL
LIN {X 0,Y 419.414,Z 444.673,A -85,B 0,C 180,E1 17651.692,E2 17651.692} C_VEL
LIN {X 0,Y 416.067,Z 440.931,A -85,B 0,C 180,E1 17649.057,E2 17649.057} C_VEL
LIN {X 0,Y 414.944,Z 438.835,A -85,B 0,C 180,E1 17647.895,E2 17647.895} C_VEL
LIN {X 0,Y 410.991,Z 434.346,A -85,B 0,C 180,E1 17641.394,E2 17641.394} C_VEL
LIN {X 0,Y 410.809,Z 433.294,A -85,B 0,C 180,E1 17639.163,E2 17639.163} C_VEL
LIN {X 0,Y 410.994,Z 434.348,A -85,B 0,C 180,E1 17636.932,E2 17636.932} C_VEL
LIN {X 0,Y 414.811,Z 438.779,A -85,B 0,C 180,E1 17630.566,E2 17630.566} C_VEL
LIN {X 0,Y 415.358,Z 439.369,A -85,B 0,C 180,E1 17630.019,E2 17630.019} C_VEL
LIN {X 0,Y 417.74,Z 443.249,A -85,B 0,C 180,E1 17627.84,E2 17627.84} C_VEL
LIN {X 0,Y 420.018,Z 445.339,A -85,B 0,C 180,E1 17626.228,E2 17626.228} C_VEL
LIN {X 0,Y 423.126,Z 449.666,A -85,B 0,C 180,E1 17624.231,E2 17624.231} C_VEL
LIN {X 0,Y 424.657,Z 451.317,A -85,B 0,C 180,E1 17623.376,E2 17623.376} C_VEL
LIN {X 0,Y 429.284,Z 457.356,A -85,B 0,C 180,E1 17621.007,E2 17621.007} C_VEL
LIN {X 0,Y 433.486,Z 462.944,A -85,B 0,C 180,E1 17619.122,E2 17619.122} C_VEL
LIN {X 0,Y 438.796,Z 471.036,A -85,B 0,C 180,E1 17616.96,E2 17616.96} C_VEL
LIN {X 0,Y 445.496,Z 481.462,A -85,B 0,C 180,E1 17614.544,E2 17614.544} C_VEL
LIN {X 0,Y 454.24,Z 495.979,A -85,B 0,C 180,E1 17611.753,E2 17611.753} C_VEL
LIN {X 0,Y 462.483,Z 510.87,A -85,B 0,C 180,E1 17609.392,E2 17609.392} C_VEL
LIN {X 0,Y 464.434,Z 514.678,A -85,B 0,C 180,E1 17608.861,E2 17608.861} C_VEL
LIN {X 0,Y 448.744,Z 755.445,A -85,B 0,C 180,E1 17604.988,E2 17604.988} C_VEL
LIN {X 0,Y 446.107,Z 780.195,A -85,B 0,C 180,E1 17604.487,E2 17604.487} C_VEL
LIN {X 0,Y 442.178,Z 804.436,A -85,B 0,C 180,E1 17603.817,E2 17603.817} C_VEL
LIN {X 0,Y 437.618,Z 827.548,A -85,B 0,C 180,E1 17602.992,E2 17602.992} C_VEL
LIN {X 0,Y 431.928,Z 850.988,A -85,B 0,C 180,E1 17601.914,E2 17601.914} C_VEL
LIN {X 0,Y 426.407,Z 871.122,A -85,B 0,C 180,E1 17600.786,E2 17600.786} C_VEL
LIN {X 0,Y 419.487,Z 893.253,A -85,B 0,C 180,E1 17599.287,E2 17599.287} C_VEL
LIN {X 0,Y 413.371,Z 911.069,A -85,B 0,C 180,E1 17597.849,E2 17597.849} C_VEL
LIN {X 0,Y 405.816,Z 931.508,A -85,B 0,C 180,E1 17595.908,E2 17595.908} C_VEL
LIN {X 0,Y 398.479,Z 949.77,A -85,B 0,C 180,E1 17593.833,E2 17593.833} C_VEL
LIN {X 0,Y 391.064,Z 967.555,A -85,B 0,C 180,E1 17591.47,E2 17591.47} C_VEL
LIN {X 0,Y 383.78,Z 984.132,A -85,B 0,C 180,E1 17588.83,E2 17588.83} C_VEL
LIN {X 0,Y 377.203,Z 999.1,A -85,B 0,C 180,E1 17586.049,E2 17586.049} C_VEL
LIN {X 0,Y 370.747,Z 1013.623,A -85,B 0,C 180,E1 17582.826,E2 17582.826} C_VEL
LIN {X 0,Y 365.59,Z 1025.702,A -85,B 0,C 180,E1 17579.672,E2 17579.672} C_VEL
LIN {X 0,Y 360.788,Z 1037.528,A -85,B 0,C 180,E1 17575.969,E2 17575.969} C_VEL
LIN {X 0,Y 357.556,Z 1046.378,A -85,B 0,C 180,E1 17572.656,E2 17572.656} C_VEL
LIN {X 0,Y 354.658,Z 1055.63,A -85,B 0,C 180,E1 17568.407,E2 17568.407} C_VEL
LIN {X 0,Y 353.183,Z 1061.621,A -85,B 0,C 180,E1 17564.929,E2 17564.929} C_VEL
LIN {X 0,Y 352.279,Z 1066.928,A -85,B 0,C 180,E1 17560.963,E2 17560.963} C_VEL
LIN {X 0,Y 351.995,Z 1070.211,A -85,B 0,C 180,E1 17557.344,E2 17557.344} C_VEL
LIN {X 0,Y 351.951,Z 1071.999,A -85,B 0,C 180,E1 17554.236,E2 17554.236} C_VEL
LIN {X 0,Y 351.973,Z 1072.815,A -85,B 0,C 180,E1 17550.977,E2 17550.977} C_VEL
LIN {X 0,Y 351.967,Z 1072.366,A -85,B 0,C 180,E1 17547.232,E2 17547.232} C_VEL
LIN {X 0,Y 351.967,Z 1070.589,A -85,B 0,C 180,E1 17543.803,E2 17543.803} C_VEL
LIN {X 0,Y 352.107,Z 1067.776,A -85,B 0,C 180,E1 17540.52,E2 17540.52} C_VEL
LIN {X 0,Y 352.731,Z 1062.919,A -85,B 0,C 180,E1 17536.559,E2 17536.559} C_VEL
LIN {X 0,Y 353.947,Z 1056.822,A -85,B 0,C 180,E1 17532.915,E2 17532.915} C_VEL
LIN {X 0,Y 355.965,Z 1049.31,A -85,B 0,C 180,E1 17529.272,E2 17529.272} C_VEL
LIN {X 0,Y 359.067,Z 1039.611,A -85,B 0,C 180,E1 17525.486,E2 17525.486} C_VEL
LIN {X 0,Y 362.686,Z 1029.662,A -85,B 0,C 180,E1 17522.231,E2 17522.231} C_VEL
LIN {X 0,Y 367.966,Z 1016.219,A -85,B 0,C 180,E1 17518.552,E2 17518.552} C_VEL
LIN {X 0,Y 373.183,Z 1003.477,A -85,B 0,C 180,E1 17515.613,E2 17515.613} C_VEL
LIN {X 0,Y 380.209,Z 986.613,A -85,B 0,C 180,E1 17512.334,E2 17512.334} C_VEL
LIN {X 0,Y 386.364,Z 971.686,A -85,B 0,C 180,E1 17509.879,E2 17509.879} C_VEL
LIN {X 0,Y 393.942,Z 952.789,A -85,B 0,C 180,E1 17507.238,E2 17507.238} C_VEL
LIN {X 0,Y 400.418,Z 935.829,A -85,B 0,C 180,E1 17505.236,E2 17505.236} C_VEL
LIN {X 0,Y 407.616,Z 916.009,A -85,B 0,C 180,E1 17503.235,E2 17503.235} C_VEL
LIN {X 0,Y 414.205,Z 896.031,A -85,B 0,C 180,E1 17501.553,E2 17501.553} C_VEL
LIN {X 0,Y 420.649,Z 875,A -85,B 0,C 180,E1 17500.058,E2 17500.058} C_VEL
LIN {X 0,Y 426.695,Z 852.212,A -85,B 0,C 180,E1 17498.732,E2 17498.732} C_VEL
LIN {X 0,Y 431.896,Z 830.071,A -85,B 0,C 180,E1 17497.676,E2 17497.676} C_VEL
LIN {X 0,Y 436.586,Z 805.872,A -85,B 0,C 180,E1 17496.773,E2 17496.773} C_VEL
LIN {X 0,Y 440.126,Z 783.489,A -85,B 0,C 180,E1 17496.128,E2 17496.128} C_VEL
LIN {X 0,Y 442.964,Z 757.691,A -85,B 0,C 180,E1 17495.575,E2 17495.575} C_VEL
LIN {X 0,Y 457.174,Z 528.912,A -85,B 0,C 180,E1 17491.86,E2 17491.86} C_VEL
LIN {X 0,Y 458.241,Z 510.448,A -85,B 0,C 180,E1 17491.543,E2 17491.543} C_VEL
LIN {X 0,Y 449.907,Z 495.126,A -85,B 0,C 180,E1 17489.38,E2 17489.38} C_VEL
LIN {X 0,Y 442.152,Z 481.656,A -85,B 0,C 180,E1 17487.181,E2 17487.181} C_VEL
LIN {X 0,Y 434.226,Z 468.876,A -85,B 0,C 180,E1 17484.705,E2 17484.705} C_VEL
LIN {X 0,Y 426.87,Z 457.577,A -85,B 0,C 180,E1 17482.119,E2 17482.119} C_VEL
LIN {X 0,Y 422.631,Z 452.038,A -85,B 0,C 180,E1 17480.497,E2 17480.497} C_VEL
LIN {X 0,Y 419.215,Z 447.562,A -85,B 0,C 180,E1 17479.073,E2 17479.073} C_VEL
LIN {X 0,Y 415.047,Z 442.231,A -85,B 0,C 180,E1 17477.164,E2 17477.164} C_VEL
LIN {X 0,Y 411.423,Z 437.457,A -85,B 0,C 180,E1 17475.289,E2 17475.289} C_VEL
LIN {X 0,Y 407.56,Z 433.226,A -85,B 0,C 180,E1 17473.045,E2 17473.045} C_VEL
LIN {X 0,Y 406.369,Z 431.211,A -85,B 0,C 180,E1 17472.217,E2 17472.217} C_VEL
LIN {X 0,Y 403.049,Z 428.102,A -85,B 0,C 180,E1 17469.784,E2 17469.784} C_VEL
LIN {X 0,Y 401.547,Z 425.1,A -85,B 0,C 180,E1 17468.304,E2 17468.304} C_VEL
LIN {X 0,Y 397.954,Z 422.286,A -85,B 0,C 180,E1 17463.89,E2 17463.89} C_VEL
LIN {X 0,Y 396.799,Z 419.017,A -85,B 0,C 180,E1 17459.278,E2 17459.278} C_VEL
LIN {X 0,Y 396.807,Z 419.157,A -85,B 0,C 180,E1 17457.978,E2 17457.978} C_VEL
LIN {X 0,Y 400.691,Z 424.725,A -85,B 0,C 180,E1 17450.085,E2 17450.085} C_VEL
LIN {X 0,Y 401.649,Z 425.352,A -85,B 0,C 180,E1 17449.166,E2 17449.166} C_VEL
LIN {X 0,Y 404.048,Z 429.334,A -85,B 0,C 180,E1 17446.985,E2 17446.985} C_VEL
LIN {X 0,Y 406.735,Z 431.719,A -85,B 0,C 180,E1 17445.114,E2 17445.114} C_VEL
LIN {X 0,Y 409.885,Z 436.086,A -85,B 0,C 180,E1 17443.124,E2 17443.124} C_VEL
LIN {X 0,Y 411.619,Z 437.865,A -85,B 0,C 180,E1 17442.177,E2 17442.177} C_VEL
LIN {X 0,Y 415.157,Z 442.327,A -85,B 0,C 180,E1 17440.368,E2 17440.368} C_VEL
LIN {X 0,Y 420.881,Z 449.647,A -85,B 0,C 180,E1 17437.806,E2 17437.806} C_VEL
LIN {X 0,Y 425.498,Z 455.738,A -85,B 0,C 180,E1 17435.975,E2 17435.975} C_VEL
LIN {X 0,Y 431.574,Z 463.827,A -85,B 0,C 180,E1 17433.809,E2 17433.809} C_VEL
LIN {X 0,Y 441.424,Z 477.827,A -85,B 0,C 180,E1 17430.707,E2 17430.707} C_VEL
LIN {X 0,Y 450.695,Z 492.011,A -85,B 0,C 180,E1 17428.128,E2 17428.128} C_VEL
LIN {X 0,Y 458.538,Z 504.882,A -85,B 0,C 180,E1 17426.14,E2 17426.14} C_VEL
LIN {X 0,Y 443.729,Z 741.836,A -85,B 0,C 180,E1 17422.306,E2 17422.306} C_VEL
LIN {X 0,Y 441.29,Z 766.307,A -85,B 0,C 180,E1 17421.787,E2 17421.787} C_VEL
LIN {X 0,Y 437.81,Z 789.774,A -85,B 0,C 180,E1 17421.093,E2 17421.093} C_VEL
LIN {X 0,Y 433.999,Z 810.733,A -85,B 0,C 180,E1 17420.309,E2 17420.309} C_VEL
LIN {X 0,Y 428.732,Z 834.62,A -85,B 0,C 180,E1 17419.183,E2 17419.183} C_VEL
LIN {X 0,Y 423.61,Z 854.622,A -85,B 0,C 180,E1 17418.033,E2 17418.033} C_VEL
LIN {X 0,Y 416.833,Z 877.841,A -85,B 0,C 180,E1 17416.421,E2 17416.421} C_VEL
LIN {X 0,Y 410.859,Z 896.225,A -85,B 0,C 180,E1 17414.891,E2 17414.891} C_VEL
LIN {X 0,Y 403.772,Z 916.375,A -85,B 0,C 180,E1 17412.922,E2 17412.922} C_VEL
LIN {X 0,Y 397.097,Z 933.804,A -85,B 0,C 180,E1 17410.895,E2 17410.895} C_VEL
LIN {X 0,Y 390.107,Z 951.336,A -85,B 0,C 180,E1 17408.524,E2 17408.524} C_VEL
LIN {X 0,Y 382.956,Z 968.211,A -85,B 0,C 180,E1 17405.793,E2 17405.793} C_VEL
LIN {X 0,Y 376.637,Z 983.099,A -85,B 0,C 180,E1 17402.972,E2 17402.972} C_VEL
LIN {X 0,Y 370.529,Z 997.207,A -85,B 0,C 180,E1 17399.771,E2 17399.771} C_VEL
LIN {X 0,Y 365.459,Z 1009.343,A -85,B 0,C 180,E1 17396.534,E2 17396.534} C_VEL
LIN {X 0,Y 361.02,Z 1020.354,A -85,B 0,C 180,E1 17392.987,E2 17392.987} C_VEL
LIN {X 0,Y 357.798,Z 1029.176,A -85,B 0,C 180,E1 17389.594,E2 17389.594} C_VEL
LIN {X 0,Y 355.037,Z 1037.749,A -85,B 0,C 180,E1 17385.518,E2 17385.518} C_VEL
LIN {X 0,Y 353.529,Z 1043.476,A -85,B 0,C 180,E1 17382.081,E2 17382.081} C_VEL
LIN {X 0,Y 352.54,Z 1048.508,A -85,B 0,C 180,E1 17378.153,E2 17378.153} C_VEL
LIN {X 0,Y 352.13,Z 1051.608,A -85,B 0,C 180,E1 17374.56,E2 17374.56} C_VEL
LIN {X 0,Y 352.007,Z 1053.352,A -85,B 0,C 180,E1 17371.302,E2 17371.302} C_VEL
LIN {X 0,Y 351.971,Z 1054.11,A -85,B 0,C 180,E1 17367.721,E2 17367.721} C_VEL
LIN {X 0,Y 352.032,Z 1053.375,A -85,B 0,C 180,E1 17363.967,E2 17363.967} C_VEL
LIN {X 0,Y 352.203,Z 1051.642,A -85,B 0,C 180,E1 17360.687,E2 17360.687} C_VEL
LIN {X 0,Y 352.745,Z 1048.383,A -85,B 0,C 180,E1 17356.893,E2 17356.893} C_VEL
LIN {X 0,Y 353.89,Z 1043.468,A -85,B 0,C 180,E1 17353.081,E2 17353.081} C_VEL
LIN {X 0,Y 355.635,Z 1037.688,A -85,B 0,C 180,E1 17349.596,E2 17349.596} C_VEL
LIN {X 0,Y 358.748,Z 1028.987,A -85,B 0,C 180,E1 17345.463,E2 17345.463} C_VEL
LIN {X 0,Y 362.176,Z 1020.487,A -85,B 0,C 180,E1 17342.188,E2 17342.188} C_VEL
LIN {X 0,Y 367.254,Z 1008.837,A -85,B 0,C 180,E1 17338.45,E2 17338.45} C_VEL
LIN {X 0,Y 372.564,Z 997.067,A -85,B 0,C 180,E1 17335.322,E2 17335.322} C_VEL
LIN {X 0,Y 378.856,Z 983.488,A -85,B 0,C 180,E1 17332.244,E2 17332.244} C_VEL
LIN {X 0,Y 384.786,Z 970.371,A -85,B 0,C 180,E1 17329.74,E2 17329.74} C_VEL
LIN {X 0,Y 386.11,Z 965.772,A -85,B 0,C 180,E1 17328.834,E2 17328.834} C_VEL
LIN {X 0,Y 386.856,Z 953.733,A -85,B 0,C 180,E1 17326.241,E2 17326.241} C_VEL
LIN {X 0,Y 388.217,Z 949.36,A -85,B 0,C 180,E1 17325.526,E2 17325.526} C_VEL
LIN {X 0,Y 395.316,Z 933.042,A -85,B 0,C 180,E1 17323.349,E2 17323.349} C_VEL
LIN {X 0,Y 403.19,Z 913.925,A -85,B 0,C 180,E1 17321.178,E2 17321.178} C_VEL
LIN {X 0,Y 410.223,Z 895.262,A -85,B 0,C 180,E1 17319.406,E2 17319.406} C_VEL
LIN {X 0,Y 417.332,Z 874.846,A -85,B 0,C 180,E1 17317.754,E2 17317.754} C_VEL
LIN {X 0,Y 423.901,Z 853.376,A -85,B 0,C 180,E1 17316.328,E2 17316.328} C_VEL
LIN {X 0,Y 429.437,Z 832.992,A -85,B 0,C 180,E1 17315.189,E2 17315.189} C_VEL
LIN {X 0,Y 435.035,Z 808.648,A -85,B 0,C 180,E1 17314.092,E2 17314.092} C_VEL
LIN {X 0,Y 439.077,Z 787.492,A -85,B 0,C 180,E1 17313.336,E2 17313.336} C_VEL
LIN {X 0,Y 442.891,Z 761.686,A -85,B 0,C 180,E1 17312.63,E2 17312.63} C_VEL
LIN {X 0,Y 445.135,Z 739.577,A -85,B 0,C 180,E1 17312.187,E2 17312.187} C_VEL
LIN {X 0,Y 460.357,Z 513.032,A -85,B 0,C 180,E1 17308.544,E2 17308.544} C_VEL
LIN {X 0,Y 452.087,Z 499.823,A -85,B 0,C 180,E1 17306.183,E2 17306.183} C_VEL
LIN {X 0,Y 444.077,Z 487.694,A -85,B 0,C 180,E1 17303.628,E2 17303.628} C_VEL
LIN {X 0,Y 436.457,Z 476.937,A -85,B 0,C 180,E1 17300.87,E2 17300.87} C_VEL
LIN {X 0,Y 432.367,Z 471.377,A -85,B 0,C 180,E1 17299.206,E2 17299.206} C_VEL
LIN {X 0,Y 429.562,Z 467.569,A -85,B 0,C 180,E1 17297.964,E2 17297.964} C_VEL
LIN {X 0,Y 426.088,Z 462.935,A -85,B 0,C 180,E1 17296.286,E2 17296.286} C_VEL
LIN {X 0,Y 422.253,Z 457.842,A -85,B 0,C 180,E1 17294.187,E2 17294.187} C_VEL
LIN {X 0,Y 418.806,Z 453.389,A -85,B 0,C 180,E1 17291.988,E2 17291.988} C_VEL
LIN {X 0,Y 417.858,Z 452.262,A -85,B 0,C 180,E1 17291.316,E2 17291.316} C_VEL
LIN {X 0,Y 414.659,Z 448.361,A -85,B 0,C 180,E1 17288.668,E2 17288.668} C_VEL
LIN {X 0,Y 413.833,Z 446.725,A -85,B 0,C 180,E1 17287.776,E2 17287.776} C_VEL
LIN {X 0,Y 409.966,Z 442.107,A -85,B 0,C 180,E1 17281.118,E2 17281.118} C_VEL
LIN {X 0,Y 409.832,Z 441.261,A -85,B 0,C 180,E1 17279.021,E2 17279.021} C_VEL
LIN {X 0,Y 410.141,Z 442.736,A -85,B 0,C 180,E1 17276.366,E2 17276.366} C_VEL
LIN {X 0,Y 413.848,Z 446.734,A -85,B 0,C 180,E1 17270.544,E2 17270.544} C_VEL
LIN {X 0,Y 416.772,Z 451.317,A -85,B 0,C 180,E1 17267.812,E2 17267.812} C_VEL
LIN {X 0,Y 418.651,Z 453.067,A -85,B 0,C 180,E1 17266.464,E2 17266.464} C_VEL
LIN {X 0,Y 421.818,Z 457.472,A -85,B 0,C 180,E1 17264.393,E2 17264.393} C_VEL
LIN {X 0,Y 423.204,Z 459.062,A -85,B 0,C 180,E1 17263.6,E2 17263.6} C_VEL
LIN {X 0,Y 427.636,Z 464.936,A -85,B 0,C 180,E1 17261.282,E2 17261.282} C_VEL
LIN {X 0,Y 431.762,Z 470.528,A -85,B 0,C 180,E1 17259.39,E2 17259.39} C_VEL
LIN {X 0,Y 438.209,Z 480.447,A -85,B 0,C 180,E1 17256.75,E2 17256.75} C_VEL
LIN {X 0,Y 444.561,Z 490.845,A -85,B 0,C 180,E1 17254.451,E2 17254.451} C_VEL
LIN {X 0,Y 452.035,Z 503.617,A -85,B 0,C 180,E1 17252.034,E2 17252.034} C_VEL
LIN {X 0,Y 459.559,Z 517.473,A -85,B 0,C 180,E1 17249.828,E2 17249.828} C_VEL
LIN {X 0,Y 460.135,Z 518.947,A -85,B 0,C 180,E1 17249.655,E2 17249.655} C_VEL
LIN {X 0,Y 444.218,Z 756.125,A -85,B 0,C 180,E1 17245.831,E2 17245.831} C_VEL
LIN {X 0,Y 441.424,Z 781.083,A -85,B 0,C 180,E1 17245.318,E2 17245.318} C_VEL
LIN {X 0,Y 437.519,Z 804.565,A -85,B 0,C 180,E1 17244.667,E2 17244.667} C_VEL
LIN {X 0,Y 432.836,Z 827.708,A -85,B 0,C 180,E1 17243.84,E2 17243.84} C_VEL
LIN {X 0,Y 427.311,Z 849.938,A -85,B 0,C 180,E1 17242.821,E2 17242.821} C_VEL
LIN {X 0,Y 421.976,Z 868.984,A -85,B 0,C 180,E1 17241.767,E2 17241.767} C_VEL
LIN {X 0,Y 414.527,Z 892.437,A -85,B 0,C 180,E1 17240.198,E2 17240.198} C_VEL
LIN {X 0,Y 407.952,Z 911.044,A -85,B 0,C 180,E1 17238.697,E2 17238.697} C_VEL
LIN {X 0,Y 400.174,Z 931.449,A -85,B 0,C 180,E1 17236.749,E2 17236.749} C_VEL
LIN {X 0,Y 393.017,Z 948.732,A -85,B 0,C 180,E1 17234.78,E2 17234.78} C_VEL
LIN {X 0,Y 385.807,Z 965.442,A -85,B 0,C 180,E1 17232.565,E2 17232.565} C_VEL
LIN {X 0,Y 377.909,Z 982.883,A -85,B 0,C 180,E1 17229.814,E2 17229.814} C_VEL
LIN {X 0,Y 371.316,Z 997.234,A -85,B 0,C 180,E1 17227.148,E2 17227.148} C_VEL
LIN {X 0,Y 364.413,Z 1012.203,A -85,B 0,C 180,E1 17223.849,E2 17223.849} C_VEL
LIN {X 0,Y 359.157,Z 1023.818,A -85,B 0,C 180,E1 17220.814,E2 17220.814} C_VEL
LIN {X 0,Y 353.965,Z 1035.972,A -85,B 0,C 180,E1 17217.052,E2 17217.052} C_VEL
LIN {X 0,Y 350.283,Z 1045.282,A -85,B 0,C 180,E1 17213.555,E2 17213.555} C_VEL
LIN {X 0,Y 347.367,Z 1053.9,A -85,B 0,C 180,E1 17209.681,E2 17209.681} C_VEL
LIN {X 0,Y 345.47,Z 1060.656,A -85,B 0,C 180,E1 17205.787,E2 17205.787} C_VEL
LIN {X 0,Y 344.491,Z 1065.534,A -85,B 0,C 180,E1 17202.233,E2 17202.233} C_VEL
LIN {X 0,Y 344.018,Z 1069.54,A -85,B 0,C 180,E1 17198.188,E2 17198.188} C_VEL
LIN {X 0,Y 343.956,Z 1071.582,A -85,B 0,C 180,E1 17194.836,E2 17194.836} C_VEL
LIN {X 0,Y 343.967,Z 1072.51,A -85,B 0,C 180,E1 17191.666,E2 17191.666} C_VEL
LIN {X 0,Y 343.971,Z 1072.443,A -85,B 0,C 180,E1 17188.501,E2 17188.501} C_VEL
LIN {X 0,Y 343.962,Z 1071.164,A -85,B 0,C 180,E1 17184.83,E2 17184.83} C_VEL
LIN {X 0,Y 344.07,Z 1068.196,A -85,B 0,C 180,E1 17180.971,E2 17180.971} C_VEL
LIN {X 0,Y 344.508,Z 1064.445,A -85,B 0,C 180,E1 17177.598,E2 17177.598} C_VEL
LIN {X 0,Y 345.679,Z 1058.425,A -85,B 0,C 180,E1 17173.533,E2 17173.533} C_VEL
LIN {X 0,Y 347.575,Z 1051.212,A -85,B 0,C 180,E1 17169.805,E2 17169.805} C_VEL
LIN {X 0,Y 350.422,Z 1042.532,A -85,B 0,C 180,E1 17166.098,E2 17166.098} C_VEL
LIN {X 0,Y 354.414,Z 1031.767,A -85,B 0,C 180,E1 17162.36,E2 17162.36} C_VEL
LIN {X 0,Y 358.922,Z 1020.654,A -85,B 0,C 180,E1 17159.097,E2 17159.097} C_VEL
LIN {X 0,Y 364.889,Z 1006.574,A -85,B 0,C 180,E1 17155.633,E2 17155.633} C_VEL
LIN {X 0,Y 370.7,Z 993.128,A -85,B 0,C 180,E1 17152.829,E2 17152.829} C_VEL
LIN {X 0,Y 378.081,Z 976.039,A -85,B 0,C 180,E1 17149.812,E2 17149.812} C_VEL
LIN {X 0,Y 384.649,Z 960.401,A -85,B 0,C 180,E1 17147.479,E2 17147.479} C_VEL
LIN {X 0,Y 392.269,Z 941.612,A -85,B 0,C 180,E1 17145.084,E2 17145.084} C_VEL
LIN {X 0,Y 399.107,Z 923.548,A -85,B 0,C 180,E1 17143.153,E2 17143.153} C_VEL
LIN {X 0,Y 406.178,Z 903.709,A -85,B 0,C 180,E1 17141.339,E2 17141.339} C_VEL
LIN {X 0,Y 413.066,Z 882.274,A -85,B 0,C 180,E1 17139.721,E2 17139.721} C_VEL
LIN {X 0,Y 418.84,Z 862.438,A -85,B 0,C 180,E1 17138.461,E2 17138.461} C_VEL
LIN {X 0,Y 424.997,Z 838.146,A -85,B 0,C 180,E1 17137.203,E2 17137.203} C_VEL
LIN {X 0,Y 429.429,Z 817.828,A -85,B 0,C 180,E1 17136.359,E2 17136.359} C_VEL
LIN {X 0,Y 433.907,Z 792.97,A -85,B 0,C 180,E1 17135.544,E2 17135.544} C_VEL
LIN {X 0,Y 436.925,Z 770.642,A -85,B 0,C 180,E1 17134.995,E2 17134.995} C_VEL
LIN {X 0,Y 439.222,Z 744.431,A -85,B 0,C 180,E1 17134.5,E2 17134.5} C_VEL
LIN {X 0,Y 453.782,Z 514.45,A -85,B 0,C 180,E1 17130.772,E2 17130.772} C_VEL
LIN {X 0,Y 445.888,Z 499.814,A -85,B 0,C 180,E1 17128.642,E2 17128.642} C_VEL
LIN {X 0,Y 439.016,Z 487.752,A -85,B 0,C 180,E1 17126.623,E2 17126.623} C_VEL
LIN {X 0,Y 431.635,Z 475.607,A -85,B 0,C 180,E1 17124.243,E2 17124.243} C_VEL
LIN {X 0,Y 424.599,Z 464.616,A -85,B 0,C 180,E1 17121.698,E2 17121.698} C_VEL
LIN {X 0,Y 420.526,Z 459.198,A -85,B 0,C 180,E1 17120.095,E2 17120.095} C_VEL
LIN {X 0,Y 417.178,Z 454.774,A -85,B 0,C 180,E1 17118.661,E2 17118.661} C_VEL
LIN {X 0,Y 413.242,Z 449.64,A -85,B 0,C 180,E1 17116.807,E2 17116.807} C_VEL
LIN {X 0,Y 409.203,Z 444.449,A -85,B 0,C 180,E1 17114.649,E2 17114.649} C_VEL
LIN {X 0,Y 405.851,Z 440.426,A -85,B 0,C 180,E1 17112.594,E2 17112.594} C_VEL
LIN {X 0,Y 404.77,Z 438.815,A -85,B 0,C 180,E1 17111.831,E2 17111.831} C_VEL
LIN {X 0,Y 401.587,Z 435.541,A -85,B 0,C 180,E1 17109.386,E2 17109.386} C_VEL
LIN {X 0,Y 400.27,Z 432.932,A -85,B 0,C 180,E1 17108.042,E2 17108.042} C_VEL
LIN {X 0,Y 396.63,Z 429.723,A -85,B 0,C 180,E1 17103.179,E2 17103.179} C_VEL
LIN {X 0,Y 395.824,Z 426.96,A -85,B 0,C 180,E1 17099.276,E2 17099.276} C_VEL
LIN {X 0,Y 395.829,Z 427.125,A -85,B 0,C 180,E1 17097.973,E2 17097.973} C_VEL
LIN {X 0,Y 399.586,Z 432.613,A -85,B 0,C 180,E1 17090.203,E2 17090.203} C_VEL
LIN {X 0,Y 400.45,Z 433.228,A -85,B 0,C 180,E1 17089.352,E2 17089.352} C_VEL
LIN {X 0,Y 402.899,Z 437.235,A -85,B 0,C 180,E1 17087.094,E2 17087.094} C_VEL
LIN {X 0,Y 405.348,Z 439.459,A -85,B 0,C 180,E1 17085.354,E2 17085.354} C_VEL
LIN {X 0,Y 408.565,Z 443.897,A -85,B 0,C 180,E1 17083.288,E2 17083.288} C_VEL
LIN {X 0,Y 410.133,Z 445.616,A -85,B 0,C 180,E1 17082.41,E2 17082.41} C_VEL
LIN {X 0,Y 413.78,Z 450.151,A -85,B 0,C 180,E1 17080.52,E2 17080.52} C_VEL
LIN {X 0,Y 419.127,Z 457.248,A -85,B 0,C 180,E1 17078.077,E2 17078.077} C_VEL
LIN {X 0,Y 423.598,Z 463.234,A -85,B 0,C 180,E1 17076.268,E2 17076.268} C_VEL
LIN {X 0,Y 429.495,Z 471.271,A -85,B 0,C 180,E1 17074.118,E2 17074.118} C_VEL
LIN {X 0,Y 438.817,Z 484.724,A -85,B 0,C 180,E1 17071.114,E2 17071.114} C_VEL
LIN {X 0,Y 447.84,Z 498.76,A -85,B 0,C 180,E1 17068.54,E2 17068.54} C_VEL
LIN {X 0,Y 454.002,Z 508.927,A -85,B 0,C 180,E1 17066.928,E2 17066.928} C_VEL
LIN {X 0,Y 438.923,Z 743.104,A -85,B 0,C 180,E1 17063.126,E2 17063.126} C_VEL
LIN {X 0,Y 436.313,Z 767.847,A -85,B 0,C 180,E1 17062.59,E2 17062.59} C_VEL
LIN {X 0,Y 432.881,Z 790.351,A -85,B 0,C 180,E1 17061.919,E2 17061.919} C_VEL
LIN {X 0,Y 428.949,Z 811.404,A -85,B 0,C 180,E1 17061.129,E2 17061.129} C_VEL
LIN {X 0,Y 423.547,Z 835.184,A -85,B 0,C 180,E1 17060.002,E2 17060.002} C_VEL
LIN {X 0,Y 418.294,Z 855.147,A -85,B 0,C 180,E1 17058.849,E2 17058.849} C_VEL
LIN {X 0,Y 411.333,Z 878.308,A -85,B 0,C 180,E1 17057.233,E2 17057.233} C_VEL
LIN {X 0,Y 405.192,Z 896.671,A -85,B 0,C 180,E1 17055.695,E2 17055.695} C_VEL
LIN {X 0,Y 397.655,Z 917.383,A -85,B 0,C 180,E1 17053.647,E2 17053.647} C_VEL
LIN {X 0,Y 390.791,Z 934.743,A -85,B 0,C 180,E1 17051.603,E2 17051.603} C_VEL
LIN {X 0,Y 383.383,Z 952.654,A -85,B 0,C 180,E1 17049.135,E2 17049.135} C_VEL
LIN {X 0,Y 376.393,Z 968.563,A -85,B 0,C 180,E1 17046.517,E2 17046.517} C_VEL
LIN {X 0,Y 369.506,Z 984.177,A -85,B 0,C 180,E1 17043.506,E2 17043.506} C_VEL
LIN {X 0,Y 363.474,Z 997.527,A -85,B 0,C 180,E1 17040.409,E2 17040.409} C_VEL
LIN {X 0,Y 358.039,Z 1010.001,A -85,B 0,C 180,E1 17037.017,E2 17037.017} C_VEL
LIN {X 0,Y 353.35,Z 1021.095,A -85,B 0,C 180,E1 17033.339,E2 17033.339} C_VEL
LIN {X 0,Y 349.871,Z 1030.252,A -85,B 0,C 180,E1 17029.708,E2 17029.708} C_VEL
LIN {X 0,Y 347.139,Z 1038.31,A -85,B 0,C 180,E1 17025.709,E2 17025.709} C_VEL
LIN {X 0,Y 345.575,Z 1043.981,A -85,B 0,C 180,E1 17022.194,E2 17022.194} C_VEL
LIN {X 0,Y 344.518,Z 1049.06,A -85,B 0,C 180,E1 17018.008,E2 17018.008} C_VEL
LIN {X 0,Y 344.132,Z 1051.951,A -85,B 0,C 180,E1 17014.499,E2 17014.499} C_VEL
LIN {X 0,Y 344.007,Z 1053.643,A -85,B 0,C 180,E1 17011.166,E2 17011.166} C_VEL
LIN {X 0,Y 343.975,Z 1054.3,A -85,B 0,C 180,E1 17007.334,E2 17007.334} C_VEL
LIN {X 0,Y 344.048,Z 1053.512,A -85,B 0,C 180,E1 17003.659,E2 17003.659} C_VEL
LIN {X 0,Y 344.246,Z 1051.729,A -85,B 0,C 180,E1 17000.301,E2 17000.301} C_VEL
LIN {X 0,Y 344.911,Z 1048.144,A -85,B 0,C 180,E1 16996.207,E2 16996.207} C_VEL
LIN {X 0,Y 346.175,Z 1043.221,A -85,B 0,C 180,E1 16992.397,E2 16992.397} C_VEL
LIN {X 0,Y 348.252,Z 1036.964,A -85,B 0,C 180,E1 16988.615,E2 16988.615} C_VEL
LIN {X 0,Y 351.392,Z 1028.741,A -85,B 0,C 180,E1 16984.734,E2 16984.734} C_VEL
LIN {X 0,Y 355.068,Z 1020.179,A -85,B 0,C 180,E1 16981.398,E2 16981.398} C_VEL
LIN {X 0,Y 360.682,Z 1007.932,A -85,B 0,C 180,E1 16977.465,E2 16977.465} C_VEL
LIN {X 0,Y 366.074,Z 996.554,A -85,B 0,C 180,E1 16974.424,E2 16974.424} C_VEL
LIN {X 0,Y 373.395,Z 981.283,A -85,B 0,C 180,E1 16971.002,E2 16971.002} C_VEL
LIN {X 0,Y 379.819,Z 967.675,A -85,B 0,C 180,E1 16968.44,E2 16968.44} C_VEL
LIN {X 0,Y 387.778,Z 950.382,A -85,B 0,C 180,E1 16965.671,E2 16965.671} C_VEL
LIN {X 0,Y 388.217,Z 949.36,A -85,B 0,C 180,E1 16965.526,E2 16965.526} C_VEL
LIN {X 0,Y 389.76,Z 944.239,A -85,B 0,C 180,E1 16964.697,E2 16964.697} C_VEL
LIN {X 0,Y 391.097,Z 931.691,A -85,B 0,C 180,E1 16962.395,E2 16962.395} C_VEL
LIN {X 0,Y 392.745,Z 926.172,A -85,B 0,C 180,E1 16961.637,E2 16961.637} C_VEL
LIN {X 0,Y 399.955,Z 908.591,A -85,B 0,C 180,E1 16959.758,E2 16959.758} C_VEL
LIN {X 0,Y 407.507,Z 888.86,A -85,B 0,C 180,E1 16957.958,E2 16957.958} C_VEL
LIN {X 0,Y 414.514,Z 868.19,A -85,B 0,C 180,E1 16956.399,E2 16956.399} C_VEL
LIN {X 0,Y 420.913,Z 847.335,A -85,B 0,C 180,E1 16955.078,E2 16955.078} C_VEL
LIN {X 0,Y 426.843,Z 824.704,A -85,B 0,C 180,E1 16953.904,E2 16953.904} C_VEL
LIN {X 0,Y 431.447,Z 804.13,A -85,B 0,C 180,E1 16953.032,E2 16953.032} C_VEL
LIN {X 0,Y 436.215,Z 777.819,A -85,B 0,C 180,E1 16952.164,E2 16952.164} C_VEL
LIN {X 0,Y 439.209,Z 755.869,A -85,B 0,C 180,E1 16951.624,E2 16951.624} C_VEL
LIN {X 0,Y 441.994,Z 723.365,A -85,B 0,C 180,E1 16951.042,E2 16951.042} C_VEL
LIN {X 0,Y 456.124,Z 517.378,A -85,B 0,C 180,E1 16947.729,E2 16947.729} C_VEL
LIN {X 0,Y 448.66,Z 505.374,A -85,B 0,C 180,E1 16945.511,E2 16945.511} C_VEL
LIN {X 0,Y 441.538,Z 494.436,A -85,B 0,C 180,E1 16943.16,E2 16943.16} C_VEL
LIN {X 0,Y 434.272,Z 483.973,A -85,B 0,C 180,E1 16940.451,E2 16940.451} C_VEL
LIN {X 0,Y 428.586,Z 475.918,A -85,B 0,C 180,E1 16938.006,E2 16938.006} C_VEL
LIN {X 0,Y 424.21,Z 470.199,A -85,B 0,C 180,E1 16935.868,E2 16935.868} C_VEL
LIN {X 0,Y 420.706,Z 465.425,A -85,B 0,C 180,E1 16933.889,E2 16933.889} C_VEL
LIN {X 0,Y 417.351,Z 460.927,A -85,B 0,C 180,E1 16931.68,E2 16931.68} C_VEL
LIN {X 0,Y 413.336,Z 455.914,A -85,B 0,C 180,E1 16928.346,E2 16928.346} C_VEL
LIN {X 0,Y 412.586,Z 454.544,A -85,B 0,C 180,E1 16927.52,E2 16927.52} C_VEL
LIN {X 0,Y 408.866,Z 449.156,A -85,B 0,C 180,E1 16919.44,E2 16919.44} C_VEL
LIN {X 0,Y 408.943,Z 449.941,A -85,B 0,C 180,E1 16917.478,E2 16917.478} C_VEL
LIN {X 0,Y 412.932,Z 454.919,A -85,B 0,C 180,E1 16910.452,E2 16910.452} C_VEL
LIN {X 0,Y 415.285,Z 458.851,A -85,B 0,C 180,E1 16908.191,E2 16908.191} C_VEL
LIN {X 0,Y 417.379,Z 460.963,A -85,B 0,C 180,E1 16906.633,E2 16906.633} C_VEL
LIN {X 0,Y 420.627,Z 465.387,A -85,B 0,C 180,E1 16904.489,E2 16904.489} C_VEL
LIN {X 0,Y 421.981,Z 467.163,A -85,B 0,C 180,E1 16903.693,E2 16903.693} C_VEL
LIN {X 0,Y 425.927,Z 472.402,A -85,B 0,C 180,E1 16901.594,E2 16901.594} C_VEL
LIN {X 0,Y 430.119,Z 478.213,A -85,B 0,C 180,E1 16899.627,E2 16899.627} C_VEL
LIN {X 0,Y 436.387,Z 488.165,A -85,B 0,C 180,E1 16897.004,E2 16897.004} C_VEL
LIN {X 0,Y 442.221,Z 497.87,A -85,B 0,C 180,E1 16894.844,E2 16894.844} C_VEL
LIN {X 0,Y 449.466,Z 510.541,A -85,B 0,C 180,E1 16892.437,E2 16892.437} C_VEL
LIN {X 0,Y 455.955,Z 522.772,A -85,B 0,C 180,E1 16890.471,E2 16890.471} C_VEL
LIN {X 0,Y 439.817,Z 756.489,A -85,B 0,C 180,E1 16886.696,E2 16886.696} C_VEL
LIN {X 0,Y 436.861,Z 781.805,A -85,B 0,C 180,E1 16886.17,E2 16886.17} C_VEL
LIN {X 0,Y 432.958,Z 804.698,A -85,B 0,C 180,E1 16885.535,E2 16885.535} C_VEL
LIN {X 0,Y 428.149,Z 827.855,A -85,B 0,C 180,E1 16884.708,E2 16884.708} C_VEL
LIN {X 0,Y 422.493,Z 850.019,A -85,B 0,C 180,E1 16883.692,E2 16883.692} C_VEL
LIN {X 0,Y 416.727,Z 870.035,A -85,B 0,C 180,E1 16882.58,E2 16882.58} C_VEL
LIN {X 0,Y 409.383,Z 892.432,A -85,B 0,C 180,E1 16881.07,E2 16881.07} C_VEL
LIN {X 0,Y 402.868,Z 910.361,A -85,B 0,C 180,E1 16879.625,E2 16879.625} C_VEL
LIN {X 0,Y 394.882,Z 930.781,A -85,B 0,C 180,E1 16877.679,E2 16877.679} C_VEL
LIN {X 0,Y 387.308,Z 948.509,A -85,B 0,C 180,E1 16875.653,E2 16875.653} C_VEL
LIN {X 0,Y 379.739,Z 965.481,A -85,B 0,C 180,E1 16873.386,E2 16873.386} C_VEL
LIN {X 0,Y 371.612,Z 982.773,A -85,B 0,C 180,E1 16870.628,E2 16870.628} C_VEL
LIN {X 0,Y 364.666,Z 997.309,A -85,B 0,C 180,E1 16867.893,E2 16867.893} C_VEL
LIN {X 0,Y 357.566,Z 1012.065,A -85,B 0,C 180,E1 16864.588,E2 16864.588} C_VEL
LIN {X 0,Y 352.066,Z 1023.671,A -85,B 0,C 180,E1 16861.505,E2 16861.505} C_VEL
LIN {X 0,Y 346.61,Z 1035.819,A -85,B 0,C 180,E1 16857.671,E2 16857.671} C_VEL
LIN {X 0,Y 342.639,Z 1045.323,A -85,B 0,C 180,E1 16854.02,E2 16854.02} C_VEL
LIN {X 0,Y 339.517,Z 1054.033,A -85,B 0,C 180,E1 16849.976,E2 16849.976} C_VEL
LIN {X 0,Y 337.534,Z 1060.729,A -85,B 0,C 180,E1 16845.992,E2 16845.992} C_VEL
LIN {X 0,Y 336.467,Z 1065.837,A -85,B 0,C 180,E1 16842.121,E2 16842.121} C_VEL
LIN {X 0,Y 336.008,Z 1069.573,A -85,B 0,C 180,E1 16838.04,E2 16838.04} C_VEL
LIN {X 0,Y 335.957,Z 1071.446,A -85,B 0,C 180,E1 16834.78,E2 16834.78} C_VEL
LIN {X 0,Y 335.971,Z 1072.323,A -85,B 0,C 180,E1 16831.535,E2 16831.535} C_VEL
LIN {X 0,Y 335.972,Z 1072.18,A -85,B 0,C 180,E1 16828.124,E2 16828.124} C_VEL
LIN {X 0,Y 335.967,Z 1070.597,A -85,B 0,C 180,E1 16824.192,E2 16824.192} C_VEL
LIN {X 0,Y 336.099,Z 1067.797,A -85,B 0,C 180,E1 16820.583,E2 16820.583} C_VEL
LIN {X 0,Y 336.6,Z 1063.99,A -85,B 0,C 180,E1 16817.127,E2 16817.127} C_VEL
LIN {X 0,Y 337.969,Z 1057.548,A -85,B 0,C 180,E1 16812.791,E2 16812.791} C_VEL
LIN {X 0,Y 339.968,Z 1050.585,A -85,B 0,C 180,E1 16809.153,E2 16809.153} C_VEL
LIN {X 0,Y 343.204,Z 1041.391,A -85,B 0,C 180,E1 16805.195,E2 16805.195} C_VEL
LIN {X 0,Y 347.415,Z 1030.66,A -85,B 0,C 180,E1 16801.461,E2 16801.461} C_VEL
LIN {X 0,Y 352.797,Z 1018.196,A -85,B 0,C 180,E1 16797.803,E2 16797.803} C_VEL
LIN {X 0,Y 358.69,Z 1004.836,A -85,B 0,C 180,E1 16794.562,E2 16794.562} C_VEL
LIN {X 0,Y 365.412,Z 990.063,A -85,B 0,C 180,E1 16791.499,E2 16791.499} C_VEL
LIN {X 0,Y 372.605,Z 973.818,A -85,B 0,C 180,E1 16788.689,E2 16788.689} C_VEL
LIN {X 0,Y 379.486,Z 957.992,A -85,B 0,C 180,E1 16786.344,E2 16786.344} C_VEL
LIN {X 0,Y 387.669,Z 938.151,A -85,B 0,C 180,E1 16783.871,E2 16783.871} C_VEL
LIN {X 0,Y 394.697,Z 920.073,A -85,B 0,C 180,E1 16781.974,E2 16781.974} C_VEL
LIN {X 0,Y 402.681,Z 897.708,A -85,B 0,C 180,E1 16780.012,E2 16780.012} C_VEL
LIN {X 0,Y 408.89,Z 878.636,A -85,B 0,C 180,E1 16778.621,E2 16778.621} C_VEL
LIN {X 0,Y 415.881,Z 854.367,A -85,B 0,C 180,E1 16777.154,E2 16777.154} C_VEL
LIN {X 0,Y 421.016,Z 833.822,A -85,B 0,C 180,E1 16776.149,E2 16776.149} C_VEL
LIN {X 0,Y 426.279,Z 809.101,A -85,B 0,C 180,E1 16775.183,E2 16775.183} C_VEL
LIN {X 0,Y 430.086,Z 786.649,A -85,B 0,C 180,E1 16774.516,E2 16774.516} C_VEL
LIN {X 0,Y 433.247,Z 761.579,A -85,B 0,C 180,E1 16773.947,E2 16773.947} C_VEL
LIN {X 0,Y 437.351,Z 701.198,A -85,B 0,C 180,E1 16772.934,E2 16772.934} C_VEL
LIN {X 0,Y 449.348,Z 518.371,A -85,B 0,C 180,E1 16769.971,E2 16769.971} C_VEL
LIN {X 0,Y 440.643,Z 502.043,A -85,B 0,C 180,E1 16767.502,E2 16767.502} C_VEL
LIN {X 0,Y 431.8,Z 486.707,A -85,B 0,C 180,E1 16764.707,E2 16764.707} C_VEL
LIN {X 0,Y 423.506,Z 473.345,A -85,B 0,C 180,E1 16761.721,E2 16761.721} C_VEL
LIN {X 0,Y 418.754,Z 466.746,A -85,B 0,C 180,E1 16759.82,E2 16759.82} C_VEL
LIN {X 0,Y 415.164,Z 461.972,A -85,B 0,C 180,E1 16758.246,E2 16758.246} C_VEL
LIN {X 0,Y 411.589,Z 457.185,A -85,B 0,C 180,E1 16756.513,E2 16756.513} C_VEL
LIN {X 0,Y 407.746,Z 452.143,A -85,B 0,C 180,E1 16754.413,E2 16754.413} C_VEL
LIN {X 0,Y 404.358,Z 447.962,A -85,B 0,C 180,E1 16752.278,E2 16752.278} C_VEL
LIN {X 0,Y 403.394,Z 446.548,A -85,B 0,C 180,E1 16751.582,E2 16751.582} C_VEL
LIN {X 0,Y 400.293,Z 443.224,A -85,B 0,C 180,E1 16749.127,E2 16749.127} C_VEL
LIN {X 0,Y 399.001,Z 440.764,A -85,B 0,C 180,E1 16747.777,E2 16747.777} C_VEL
LIN {X 0,Y 395.27,Z 436.942,A -85,B 0,C 180,E1 16742.175,E2 16742.175} C_VEL
LIN {X 0,Y 394.845,Z 434.875,A -85,B 0,C 180,E1 16739.129,E2 16739.129} C_VEL
LIN {X 0,Y 394.857,Z 435.17,A -85,B 0,C 180,E1 16737.823,E2 16737.823} C_VEL
LIN {X 0,Y 398.484,Z 440.502,A -85,B 0,C 180,E1 16730.321,E2 16730.321} C_VEL
LIN {X 0,Y 399.32,Z 441.244,A -85,B 0,C 180,E1 16729.468,E2 16729.468} C_VEL
LIN {X 0,Y 401.931,Z 445.323,A -85,B 0,C 180,E1 16727.062,E2 16727.062} C_VEL
LIN {X 0,Y 403.969,Z 447.193,A -85,B 0,C 180,E1 16725.596,E2 16725.596} C_VEL
LIN {X 0,Y 407.247,Z 451.707,A -85,B 0,C 180,E1 16723.453,E2 16723.453} C_VEL
LIN {X 0,Y 408.559,Z 453.198,A -85,B 0,C 180,E1 16722.701,E2 16722.701} C_VEL
LIN {X 0,Y 413.123,Z 459.198,A -85,B 0,C 180,E1 16720.305,E2 16720.305} C_VEL
LIN {X 0,Y 417.384,Z 464.843,A -85,B 0,C 180,E1 16718.351,E2 16718.351} C_VEL
LIN {X 0,Y 421.791,Z 470.84,A -85,B 0,C 180,E1 16716.531,E2 16716.531} C_VEL
LIN {X 0,Y 427.518,Z 478.842,A -85,B 0,C 180,E1 16714.399,E2 16714.399} C_VEL
LIN {X 0,Y 436.232,Z 491.621,A -85,B 0,C 180,E1 16711.526,E2 16711.526} C_VEL
LIN {X 0,Y 445.114,Z 505.677,A -85,B 0,C 180,E1 16708.929,E2 16708.929} C_VEL
LIN {X 0,Y 449.528,Z 513.335,A -85,B 0,C 180,E1 16707.726,E2 16707.726} C_VEL
LIN {X 0,Y 434.242,Z 743.941,A -85,B 0,C 180,E1 16703.971,E2 16703.971} C_VEL
LIN {X 0,Y 431.442,Z 769.257,A -85,B 0,C 180,E1 16703.414,E2 16703.414} C_VEL
LIN {X 0,Y 428.047,Z 790.905,A -85,B 0,C 180,E1 16702.765,E2 16702.765} C_VEL
LIN {X 0,Y 423.703,Z 813.538,A -85,B 0,C 180,E1 16701.908,E2 16701.908} C_VEL
LIN {X 0,Y 418.451,Z 835.747,A -85,B 0,C 180,E1 16700.841,E2 16700.841} C_VEL
LIN {X 0,Y 413.066,Z 855.673,A -85,B 0,C 180,E1 16699.686,E2 16699.686} C_VEL
LIN {X 0,Y 405.918,Z 878.775,A -85,B 0,C 180,E1 16698.066,E2 16698.066} C_VEL
LIN {X 0,Y 399.591,Z 897.159,A -85,B 0,C 180,E1 16696.517,E2 16696.517} C_VEL
LIN {X 0,Y 391.848,Z 917.789,A -85,B 0,C 180,E1 16694.463,E2 16694.463} C_VEL
LIN {X 0,Y 384.794,Z 935.08,A -85,B 0,C 180,E1 16692.411,E2 16692.411} C_VEL
LIN {X 0,Y 377.123,Z 953.017,A -85,B 0,C 180,E1 16689.913,E2 16689.913} C_VEL
LIN {X 0,Y 369.893,Z 968.914,A -85,B 0,C 180,E1 16687.266,E2 16687.266} C_VEL
LIN {X 0,Y 362.722,Z 984.541,A -85,B 0,C 180,E1 16684.209,E2 16684.209} C_VEL
LIN {X 0,Y 356.465,Z 997.846,A -85,B 0,C 180,E1 16681.073,E2 16681.073} C_VEL
LIN {X 0,Y 350.875,Z 1010.119,A -85,B 0,C 180,E1 16677.678,E2 16677.678} C_VEL
LIN {X 0,Y 346.08,Z 1020.937,A -85,B 0,C 180,E1 16674.04,E2 16674.04} C_VEL
LIN {X 0,Y 342.51,Z 1029.741,A -85,B 0,C 180,E1 16670.507,E2 16670.507} C_VEL
LIN {X 0,Y 339.439,Z 1038.279,A -85,B 0,C 180,E1 16666.251,E2 16666.251} C_VEL
LIN {X 0,Y 337.744,Z 1043.99,A -85,B 0,C 180,E1 16662.655,E2 16662.655} C_VEL
LIN {X 0,Y 336.591,Z 1049.144,A -85,B 0,C 180,E1 16658.37,E2 16658.37} C_VEL
LIN {X 0,Y 336.153,Z 1052.073,A -85,B 0,C 180,E1 16654.777,E2 16654.777} C_VEL
LIN {X 0,Y 336.015,Z 1053.801,A -85,B 0,C 180,E1 16651.364,E2 16651.364} C_VEL
LIN {X 0,Y 335.977,Z 1054.542,A -85,B 0,C 180,E1 16647.612,E2 16647.612} C_VEL
LIN {X 0,Y 336.051,Z 1053.782,A -85,B 0,C 180,E1 16643.679,E2 16643.679} C_VEL
LIN {X 0,Y 336.257,Z 1052.037,A -85,B 0,C 180,E1 16640.242,E2 16640.242} C_VEL
LIN {X 0,Y 336.905,Z 1048.765,A -85,B 0,C 180,E1 16636.265,E2 16636.265} C_VEL
LIN {X 0,Y 338.233,Z 1043.823,A -85,B 0,C 180,E1 16632.272,E2 16632.272} C_VEL
LIN {X 0,Y 340.229,Z 1038.029,A -85,B 0,C 180,E1 16628.628,E2 16628.628} C_VEL
LIN {X 0,Y 343.756,Z 1029.296,A -85,B 0,C 180,E1 16624.317,E2 16624.317} C_VEL
LIN {X 0,Y 347.805,Z 1020.326,A -85,B 0,C 180,E1 16620.743,E2 16620.743} C_VEL
LIN {X 0,Y 353.711,Z 1008.06,A -85,B 0,C 180,E1 16616.742,E2 16616.742} C_VEL
LIN {X 0,Y 359.355,Z 996.673,A -85,B 0,C 180,E1 16613.654,E2 16613.654} C_VEL
LIN {X 0,Y 366.994,Z 981.38,A -85,B 0,C 180,E1 16610.188,E2 16610.188} C_VEL
LIN {X 0,Y 373.667,Z 967.759,A -85,B 0,C 180,E1 16607.598,E2 16607.598} C_VEL
LIN {X 0,Y 381.915,Z 950.439,A -85,B 0,C 180,E1 16604.805,E2 16604.805} C_VEL
LIN {X 0,Y 389.183,Z 934.285,A -85,B 0,C 180,E1 16602.62,E2 16602.62} C_VEL
LIN {X 0,Y 392.745,Z 926.172,A -85,B 0,C 180,E1 16601.637,E2 16601.637} C_VEL
LIN {X 0,Y 394.432,Z 920.552,A -85,B 0,C 180,E1 16600.895,E2 16600.895} C_VEL
LIN {X 0,Y 396.226,Z 906.857,A -85,B 0,C 180,E1 16598.774,E2 16598.774} C_VEL
LIN {X 0,Y 397.893,Z 900.897,A -85,B 0,C 180,E1 16598.1,E2 16598.1} C_VEL
LIN {X 0,Y 405.199,Z 881.272,A -85,B 0,C 180,E1 16596.442,E2 16596.442} C_VEL
LIN {X 0,Y 412.345,Z 860.319,A -85,B 0,C 180,E1 16594.954,E2 16594.954} C_VEL
LIN {X 0,Y 418.746,Z 838.389,A -85,B 0,C 180,E1 16593.679,E2 16593.679} C_VEL
LIN {X 0,Y 424.105,Z 817.533,A -85,B 0,C 180,E1 16592.677,E2 16592.677} C_VEL
LIN {X 0,Y 429.224,Z 793.283,A -85,B 0,C 180,E1 16591.751,E2 16591.751} C_VEL
LIN {X 0,Y 432.677,Z 772.93,A -85,B 0,C 180,E1 16591.14,E2 16591.14} C_VEL
LIN {X 0,Y 435.925,Z 747.159,A -85,B 0,C 180,E1 16590.558,E2 16590.558} C_VEL
LIN {X 0,Y 442.486,Z 655.849,A -85,B 0,C 180,E1 16589.06,E2 16589.06} C_VEL
LIN {X 0,Y 452.005,Z 521.752,A -85,B 0,C 180,E1 16586.904,E2 16586.904} C_VEL
LIN {X 0,Y 443.659,Z 508.27,A -85,B 0,C 180,E1 16584.287,E2 16584.287} C_VEL
LIN {X 0,Y 436.155,Z 496.857,A -85,B 0,C 180,E1 16581.625,E2 16581.625} C_VEL
LIN {X 0,Y 429.722,Z 487.543,A -85,B 0,C 180,E1 16579.012,E2 16579.012} C_VEL
LIN {X 0,Y 425.663,Z 481.958,A -85,B 0,C 180,E1 16577.146,E2 16577.146} C_VEL
LIN {X 0,Y 422.605,Z 477.743,A -85,B 0,C 180,E1 16575.578,E2 16575.578} C_VEL
LIN {X 0,Y 419.172,Z 473.003,A -85,B 0,C 180,E1 16573.589,E2 16573.589} C_VEL
LIN {X 0,Y 415.354,Z 467.868,A -85,B 0,C 180,E1 16570.963,E2 16570.963} C_VEL
LIN {X 0,Y 412.211,Z 463.859,A -85,B 0,C 180,E1 16568.228,E2 16568.228} C_VEL
LIN {X 0,Y 411.481,Z 462.432,A -85,B 0,C 180,E1 16567.4,E2 16567.4} C_VEL
LIN {X 0,Y 407.888,Z 457.115,A -85,B 0,C 180,E1 16559.438,E2 16559.438} C_VEL
LIN {X 0,Y 407.965,Z 457.915,A -85,B 0,C 180,E1 16557.471,E2 16557.471} C_VEL
LIN {X 0,Y 411.813,Z 462.908,A -85,B 0,C 180,E1 16550.567,E2 16550.567} C_VEL
LIN {X 0,Y 414.315,Z 466.922,A -85,B 0,C 180,E1 16548.163,E2 16548.163} C_VEL
LIN {X 0,Y 416.026,Z 468.681,A -85,B 0,C 180,E1 16546.872,E2 16546.872} C_VEL
LIN {X 0,Y 419.324,Z 473.192,A -85,B 0,C 180,E1 16544.652,E2 16544.652} C_VEL
LIN {X 0,Y 424.169,Z 479.768,A -85,B 0,C 180,E1 16541.942,E2 16541.942} C_VEL
LIN {X 0,Y 428.555,Z 485.995,A -85,B 0,C 180,E1 16539.835,E2 16539.835} C_VEL
LIN {X 0,Y 435.127,Z 496.806,A -85,B 0,C 180,E1 16537.041,E2 16537.041} C_VEL
LIN {X 0,Y 440.33,Z 505.638,A -85,B 0,C 180,E1 16535.088,E2 16535.088} C_VEL
LIN {X 0,Y 447.477,Z 518.495,A -85,B 0,C 180,E1 16532.665,E2 16532.665} C_VEL
LIN {X 0,Y 451.836,Z 527.059,A -85,B 0,C 180,E1 16531.294,E2 16531.294} C_VEL
LIN {X 0,Y 435.519,Z 756.853,A -85,B 0,C 180,E1 16527.578,E2 16527.578} C_VEL
LIN {X 0,Y 432.354,Z 782.787,A -85,B 0,C 180,E1 16527.034,E2 16527.034} C_VEL
LIN {X 0,Y 428.457,Z 805.047,A -85,B 0,C 180,E1 16526.414,E2 16526.414} C_VEL
LIN {X 0,Y 423.561,Z 827.986,A -85,B 0,C 180,E1 16525.594,E2 16525.594} C_VEL
LIN {X 0,Y 417.776,Z 850.1,A -85,B 0,C 180,E1 16524.582,E2 16524.582} C_VEL
LIN {X 0,Y 411.866,Z 870.084,A -85,B 0,C 180,E1 16523.472,E2 16523.472} C_VEL
LIN {X 0,Y 404.337,Z 892.43,A -85,B 0,C 180,E1 16521.964,E2 16521.964} C_VEL
LIN {X 0,Y 397.403,Z 910.965,A -85,B 0,C 180,E1 16520.464,E2 16520.464} C_VEL
LIN {X 0,Y 388.89,Z 931.941,A -85,B 0,C 180,E1 16518.435,E2 16518.435} C_VEL
LIN {X 0,Y 381.372,Z 948.993,A -85,B 0,C 180,E1 16516.463,E2 16516.463} C_VEL
LIN {X 0,Y 373.171,Z 966.79,A -85,B 0,C 180,E1 16514.052,E2 16514.052} C_VEL
LIN {X 0,Y 364.97,Z 983.514,A -85,B 0,C 180,E1 16511.319,E2 16511.319} C_VEL
LIN {X 0,Y 357.431,Z 998.739,A -85,B 0,C 180,E1 16508.391,E2 16508.391} C_VEL
LIN {X 0,Y 350.129,Z 1013.207,A -85,B 0,C 180,E1 16505.03,E2 16505.03} C_VEL
LIN {X 0,Y 344.046,Z 1025.609,A -85,B 0,C 180,E1 16501.62,E2 16501.62} C_VEL
LIN {X 0,Y 338.647,Z 1037.043,A -85,B 0,C 180,E1 16497.808,E2 16497.808} C_VEL
LIN {X 0,Y 334.699,Z 1046.177,A -85,B 0,C 180,E1 16494.16,E2 16494.16} C_VEL
LIN {X 0,Y 331.349,Z 1055.087,A -85,B 0,C 180,E1 16489.754,E2 16489.754} C_VEL
LIN {X 0,Y 329.535,Z 1061.062,A -85,B 0,C 180,E1 16486.029,E2 16486.029} C_VEL
LIN {X 0,Y 328.402,Z 1066.337,A -85,B 0,C 180,E1 16481.771,E2 16481.771} C_VEL
LIN {X 0,Y 327.999,Z 1069.606,A -85,B 0,C 180,E1 16477.885,E2 16477.885} C_VEL
LIN {X 0,Y 327.956,Z 1071.381,A -85,B 0,C 180,E1 16474.547,E2 16474.547} C_VEL
LIN {X 0,Y 327.98,Z 1072.183,A -85,B 0,C 180,E1 16471.048,E2 16471.048} C_VEL
LIN {X 0,Y 327.973,Z 1071.769,A -85,B 0,C 180,E1 16467.204,E2 16467.204} C_VEL
LIN {X 0,Y 327.969,Z 1070.019,A -85,B 0,C 180,E1 16463.523,E2 16463.523} C_VEL
LIN {X 0,Y 328.157,Z 1067.233,A -85,B 0,C 180,E1 16459.998,E2 16459.998} C_VEL
LIN {X 0,Y 328.882,Z 1062.645,A -85,B 0,C 180,E1 16455.895,E2 16455.895} C_VEL
LIN {X 0,Y 330.391,Z 1056.359,A -85,B 0,C 180,E1 16451.837,E2 16451.837} C_VEL
LIN {X 0,Y 332.654,Z 1049.236,A -85,B 0,C 180,E1 16448.117,E2 16448.117} C_VEL
LIN {X 0,Y 336.421,Z 1039.239,A -85,B 0,C 180,E1 16443.904,E2 16443.904} C_VEL
LIN {X 0,Y 340.613,Z 1029.322,A -85,B 0,C 180,E1 16440.451,E2 16440.451} C_VEL
LIN {X 0,Y 346.643,Z 1015.952,A -85,B 0,C 180,E1 16436.569,E2 16436.569} C_VEL
LIN {X 0,Y 352.292,Z 1003.81,A -85,B 0,C 180,E1 16433.616,E2 16433.616} C_VEL
LIN {X 0,Y 359.525,Z 988.495,A -85,B 0,C 180,E1 16430.44,E2 16430.44} C_VEL
LIN {X 0,Y 366.846,Z 972.536,A -85,B 0,C 180,E1 16427.683,E2 16427.683} C_VEL
LIN {X 0,Y 374.779,Z 954.924,A -85,B 0,C 180,E1 16425.09,E2 16425.09} C_VEL
LIN {X 0,Y 382.708,Z 936.061,A -85,B 0,C 180,E1 16422.789,E2 16422.789} C_VEL
LIN {X 0,Y 390.624,Z 916.247,A -85,B 0,C 180,E1 16420.74,E2 16420.74} C_VEL
LIN {X 0,Y 398.069,Z 895.555,A -85,B 0,C 180,E1 16418.975,E2 16418.975} C_VEL
LIN {X 0,Y 405.041,Z 874.546,A -85,B 0,C 180,E1 16417.471,E2 16417.471} C_VEL
LIN {X 0,Y 411.328,Z 852.711,A -85,B 0,C 180,E1 16416.191,E2 16416.191} C_VEL
LIN {X 0,Y 416.631,Z 831.84,A -85,B 0,C 180,E1 16415.185,E2 16415.185} C_VEL
LIN {X 0,Y 422.047,Z 806.369,A -85,B 0,C 180,E1 16414.218,E2 16414.218} C_VEL
LIN {X 0,Y 425.79,Z 784.423,A -85,B 0,C 180,E1 16413.582,E2 16413.582} C_VEL
LIN {X 0,Y 429.024,Z 757.571,A -85,B 0,C 180,E1 16412.998,E2 16412.998} C_VEL
LIN {X 0,Y 444.382,Z 531.076,A -85,B 0,C 180,E1 16409.292,E2 16409.292} C_VEL
LIN {X 0,Y 444.913,Z 522.26,A -85,B 0,C 180,E1 16409.133,E2 16409.133} C_VEL
LIN {X 0,Y 436.81,Z 506.792,A -85,B 0,C 180,E1 16406.731,E2 16406.731} C_VEL
LIN {X 0,Y 427.783,Z 491.002,A -85,B 0,C 180,E1 16403.742,E2 16403.742} C_VEL
LIN {X 0,Y 420.29,Z 478.9,A -85,B 0,C 180,E1 16400.907,E2 16400.907} C_VEL
LIN {X 0,Y 414.338,Z 470.487,A -85,B 0,C 180,E1 16398.356,E2 16398.356} C_VEL
LIN {X 0,Y 409.552,Z 464.294,A -85,B 0,C 180,E1 16396.015,E2 16396.015} C_VEL
LIN {X 0,Y 406.178,Z 459.729,A -85,B 0,C 180,E1 16394.106,E2 16394.106} C_VEL
LIN {X 0,Y 402.878,Z 455.499,A -85,B 0,C 180,E1 16391.96,E2 16391.96} C_VEL
LIN {X 0,Y 402.026,Z 454.278,A -85,B 0,C 180,E1 16391.331,E2 16391.331} C_VEL
LIN {X 0,Y 398.936,Z 450.781,A -85,B 0,C 180,E1 16388.794,E2 16388.794} C_VEL
LIN {X 0,Y 397.885,Z 448.657,A -85,B 0,C 180,E1 16387.654,E2 16387.654} C_VEL
LIN {X 0,Y 394.206,Z 444.697,A -85,B 0,C 180,E1 16381.89,E2 16381.89} C_VEL
LIN {X 0,Y 393.868,Z 442.79,A -85,B 0,C 180,E1 16378.982,E2 16378.982} C_VEL
LIN {X 0,Y 393.946,Z 443.622,A -85,B 0,C 180,E1 16377.042,E2 16377.042} C_VEL
LIN {X 0,Y 397.248,Z 448.311,A -85,B 0,C 180,E1 16370.584,E2 16370.584} C_VEL
LIN {X 0,Y 398.131,Z 449.096,A -85,B 0,C 180,E1 16369.655,E2 16369.655} C_VEL
LIN {X 0,Y 400.964,Z 453.399,A -85,B 0,C 180,E1 16367.03,E2 16367.03} C_VEL
LIN {X 0,Y 402.689,Z 455.096,A -85,B 0,C 180,E1 16365.77,E2 16365.77} C_VEL
LIN {X 0,Y 406.051,Z 459.628,A -85,B 0,C 180,E1 16363.55,E2 16363.55} C_VEL
LIN {X 0,Y 407.763,Z 461.997,A -85,B 0,C 180,E1 16362.541,E2 16362.541} C_VEL
LIN {X 0,Y 411.333,Z 466.572,A -85,B 0,C 180,E1 16360.658,E2 16360.658} C_VEL
LIN {X 0,Y 415.725,Z 472.537,A -85,B 0,C 180,E1 16358.593,E2 16358.593} C_VEL
LIN {X 0,Y 421.481,Z 480.366,A -85,B 0,C 180,E1 16356.215,E2 16356.215} C_VEL
LIN {X 0,Y 430.54,Z 493.714,A -85,B 0,C 180,E1 16352.96,E2 16352.96} C_VEL
LIN {X 0,Y 439.319,Z 507.498,A -85,B 0,C 180,E1 16350.215,E2 16350.215} C_VEL
LIN {X 0,Y 445.169,Z 517.392,A -85,B 0,C 180,E1 16348.546,E2 16348.546} C_VEL
LIN {X 0,Y 429.649,Z 744.88,A -85,B 0,C 180,E1 16344.833,E2 16344.833} C_VEL
LIN {X 0,Y 426.548,Z 771.399,A -85,B 0,C 180,E1 16344.237,E2 16344.237} C_VEL
LIN {X 0,Y 423.15,Z 792.357,A -85,B 0,C 180,E1 16343.599,E2 16343.599} C_VEL
LIN {X 0,Y 418.528,Z 815.533,A -85,B 0,C 180,E1 16342.708,E2 16342.708} C_VEL
LIN {X 0,Y 413.155,Z 837.428,A -85,B 0,C 180,E1 16341.64,E2 16341.64} C_VEL
LIN {X 0,Y 407.082,Z 859.179,A -85,B 0,C 180,E1 16340.357,E2 16340.357} C_VEL
LIN {X 0,Y 400.317,Z 880.043,A -85,B 0,C 180,E1 16338.857,E2 16338.857} C_VEL
LIN {X 0,Y 393.997,Z 897.864,A -85,B 0,C 180,E1 16337.344,E2 16337.344} C_VEL
LIN {X 0,Y 385.872,Z 918.795,A -85,B 0,C 180,E1 16335.235,E2 16335.235} C_VEL
LIN {X 0,Y 378.903,Z 935.352,A -85,B 0,C 180,E1 16333.252,E2 16333.252} C_VEL
LIN {X 0,Y 370.934,Z 953.38,A -85,B 0,C 180,E1 16330.718,E2 16330.718} C_VEL
LIN {X 0,Y 363.458,Z 969.265,A -85,B 0,C 180,E1 16328.042,E2 16328.042} C_VEL
LIN {X 0,Y 356.382,Z 984.12,A -85,B 0,C 180,E1 16325.111,E2 16325.111} C_VEL
LIN {X 0,Y 349.727,Z 997.709,A -85,B 0,C 180,E1 16321.881,E2 16321.881} C_VEL
LIN {X 0,Y 343.928,Z 1009.865,A -85,B 0,C 180,E1 16318.476,E2 16318.476} C_VEL
LIN {X 0,Y 338.655,Z 1021.228,A -85,B 0,C 180,E1 16314.602,E2 16314.602} C_VEL
LIN {X 0,Y 334.898,Z 1030.023,A -85,B 0,C 180,E1 16310.994,E2 16310.994} C_VEL
LIN {X 0,Y 331.657,Z 1038.544,A -85,B 0,C 180,E1 16306.643,E2 16306.643} C_VEL
LIN {X 0,Y 329.864,Z 1044.246,A -85,B 0,C 180,E1 16302.962,E2 16302.962} C_VEL
LIN {X 0,Y 328.633,Z 1049.39,A -85,B 0,C 180,E1 16298.567,E2 16298.567} C_VEL
LIN {X 0,Y 328.166,Z 1052.305,A -85,B 0,C 180,E1 16294.894,E2 16294.894} C_VEL
